# B&R Automation Studio project AP124
Automation Studio 4.2.8.54 SP; technology packages: mapp 1.40.0, TextSystem 

## Configuration CP1583

CPU X20CP1583, AutomationRuntime A4.26, Build 4.1.2, Vc V4.26.1, Safety 1.9

### Task classes (Cpu.sw)
```
Cyclic#3 (cycle 50000 us, tolerance 50000 us):
  pallet_mag <- plc.pallet_magazine.pallet_magazine.prg
  pallet_con <- plc.palletization.pallet_conveyors.pallet_conveyors.prg
  product_in <- plc.palletization.product_infeed.product_infeed.prg
  robot_head <- plc.palletization.robot_head.robot_head.prg
  robot_cont <- plc.palletization.robot_control.robot_control.prg
  wrapper <- plc.pallet_outfeed.wrapper.wrapper.prg
  pallet_out <- plc.pallet_outfeed.pallet_outfeed.pallet_outfeed.prg
  alarm_mana <- plc.alarm_management.alarm_management.prg
  safety <- safety.safety.prg
Cyclic#4 (cycle 100000 us, tolerance 100000 us):
  visu_manag <- visualization.visu_manager.prg
  visu_roman <- visualization.visu_roman.prg
DataObjects: assl1
VcDataObjects: Visu <- visualization.Visu.dob
Binaries: TCData, vcctext, arialbd, vcmgr, vccshape, vcnet, Visu02, vcbclass, vcfntttf, vctcal, Visu03, vcshared, vcrt, vcpkat, Visu01, vccbmp, vcfile, vccbtn, vccdt, vcalarm, vccnum, vcchspot, vcpdsw, vcdsint, arial, vccovl, udbdef, vccline, vcpdvnc, vccalarm, vccstr, vcchtml, vcxml, vcgclass, vccurl, vcdsloc, vcpfx20, sysconf, ashwd, asfw, iomap, Role, User, arconfig, TC, vcclbox, vcpfar00, vccscale, vccslider, arsvcreg
Libraries: AsSafety, FileIO, AsXml, standard, runtime, astime, asieccon, asstring, ashw, dataobj, vcresman, MTBasics, brsystem, MTTypes, sys_lib, AsBrStr, AcpInoSdc, AsIOAcc, AsBrMath, AsEPL, visapi
```

### Hardware
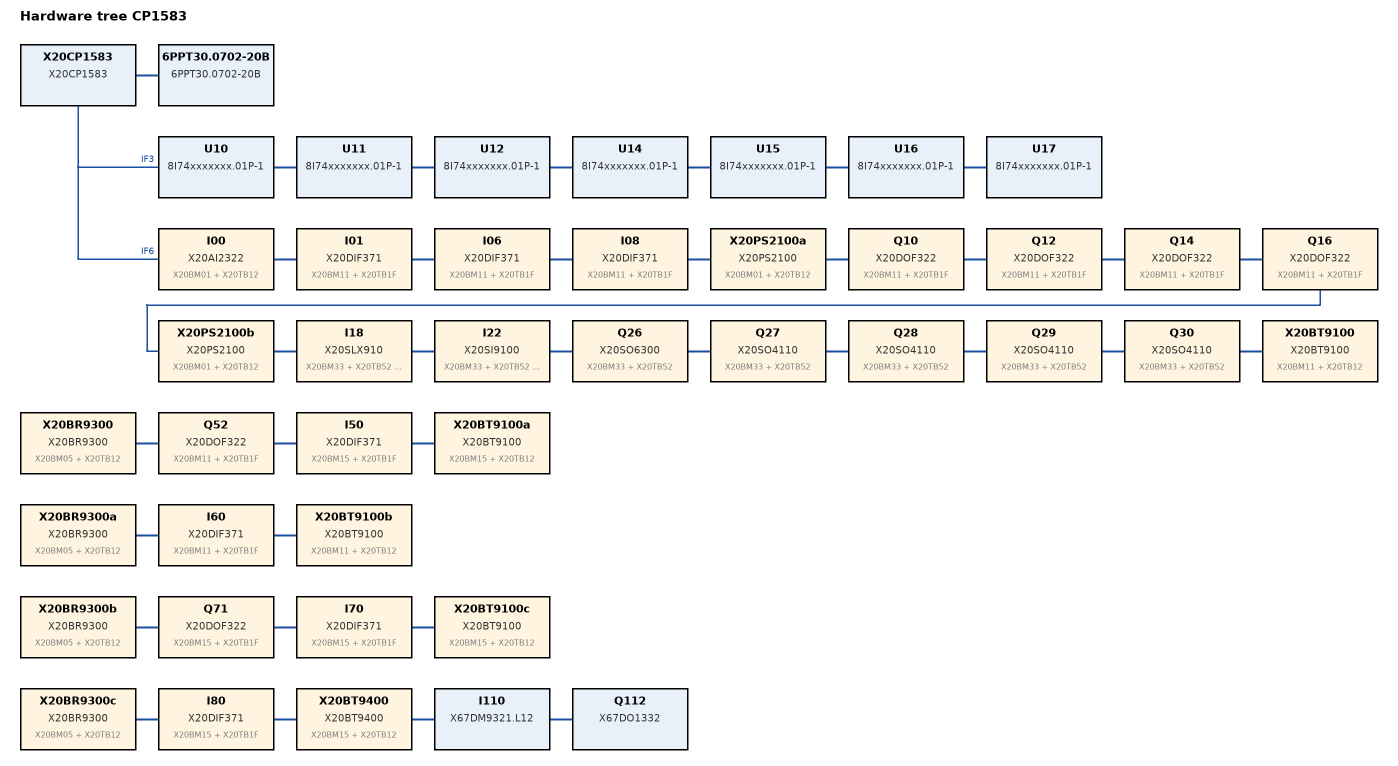
```
6PPT30.0702-20B : 6PPT30.0702-20B v1.1.0.0  [ETH1 -> X20CP1583.IF2 (NodeNumber=1)]
  Terminal = true
  Startmode = 1
  Mode = Manual
  InternetAddress = 192.168.88.11
  DefaultGateway = 192.168.88.1
  Subnetmask = 255.255.255.0
  ActivateOpenService = 0
  SelectedFavoriteVNC = 192.168.88.10
  PasswordVNC = 
  PasswordCIFS = 
  PasswordService = 
I00 : X20AI2322 v1.0.0.2  [SS1 -> X20TB12.SS; SL -> X20BM01.SL1]
  ChannelType01 = 4 to 20mA
I01 : X20DIF371 v1.0.1.0  [SS1 -> X20TB1F12.SS; SL -> X20BM11q.SL1]
I06 : X20DIF371 v1.0.1.0  [SS1 -> X20TB1F.SS; SL -> X20BM11.SL1]
I08 : X20DIF371 v1.0.1.0  [SS1 -> X20TB1F1.SS; SL -> X20BM11a.SL1]
I110 : X67DM9321.L12 v1.1.1.1 (Disabled=true)  [X2X1 -> X20BT9400.X2X1 (NodeNumber=33)]
I18 : X20SLX910 v1.10.0.0  [SS1 -> X20TB52.SS; SS2 -> X20TB52a.SS; SL -> X20BM33.SL1]
  SafeProject = SafeLOGIC-1
  SafeDesigner = 4.2.0.17
  UnsafeOutputBOOLs = 24
  UnsafeInputBOOLs = 24
I22 : X20SI9100 v1.10.0.1  [SS1 -> X20TB52b.SS; SS2 -> X20TB52c.SS; SL -> X20BM33a.SL1]
I50 : X20DIF371 v1.0.1.0  [SS1 -> X20TB1F6.SS; SL -> X20BM15f.SL1]
I60 : X20DIF371 v1.0.1.0  [SS1 -> X20TB1F8.SS; SL -> X20BM11j.SL1]
I70 : X20DIF371 v1.0.1.0  [SS1 -> X20TB1F9.SS; SL -> X20BM15c.SL1]
I80 : X20DIF371 v1.0.1.0  [SS1 -> X20TB1F11.SS; SL -> X20BM15a.SL1]
Q10 : X20DOF322 v1.1.0.2  [SS1 -> X20TB1F2.SS; SL -> X20BM11b.SL1]
Q112 : X67DO1332 v1.0.0.2 (Disabled=true)  [X2X1 -> I110.X2X2]
Q12 : X20DOF322 v1.1.0.2  [SS1 -> X20TB1F3.SS; SL -> X20BM11c.SL1]
Q14 : X20DOF322 v1.1.0.2  [SS1 -> X20TB1F4.SS; SL -> X20BM11d.SL1]
Q16 : X20DOF322 v1.1.0.2  [SS1 -> X20TB1F5.SS; SL -> X20BM11e.SL1]
Q26 : X20SO6300 v1.10.0.1  [SS1 -> X20TB52d.SS; SL -> X20BM33b.SL1]
  SafeModuleID = 3
  DigitalOutput01 = viaSafeLOGIC
  DigitalOutput02 = viaSafeLOGIC
  DigitalOutput03 = viaSafeLOGIC
  DigitalOutput04 = viaSafeLOGIC
  DigitalOutput05 = viaSafeLOGIC
  DigitalOutput06 = viaSafeLOGIC
Q27 : X20SO4110 v1.10.0.1  [SS1 -> X20TB52e.SS; SL -> X20BM33c.SL1]
  SafeModuleID = 4
Q28 : X20SO4110 v1.10.0.1  [SS1 -> X20TB52f.SS; SL -> X20BM33d.SL1]
  SafeModuleID = 5
Q29 : X20SO4110 v1.10.0.1  [SS1 -> X20TB52g.SS; SL -> X20BM33e.SL1]
  SafeModuleID = 6
  DigitalOutput01 = viaSafeLOGIC
  DigitalOutput02 = viaSafeLOGIC
  DigitalOutput03 = viaSafeLOGIC
  DigitalOutput04 = viaSafeLOGIC
Q30 : X20SO4110 v1.10.0.1  [SS1 -> X20TB52h.SS; SL -> X20BM33f.SL1]
  SafeModuleID = 7
  DigitalOutput01 = viaSafeLOGIC
  DigitalOutput02 = viaSafeLOGIC
  DigitalOutput03 = viaSafeLOGIC
  DigitalOutput04 = viaSafeLOGIC
Q52 : X20DOF322 v1.1.0.2  [SS1 -> X20TB1F7.SS; SL -> X20BM11h.SL1]
Q71 : X20DOF322 v1.1.0.2  [SS1 -> X20TB1F10.SS; SL -> X20BM15d.SL1]
U10 : 8I74xxxxxxx.01P-1 v1.3.0.0  [PLK1 -> X20CP1583.IF3 (NodeNumber=10); PLK2 -> U11.PLK1 (NodeNumber=10)]
  Supervision = off
  packedETAD = packed
  packedETI = packed
  packedCMDD = packed
  packedCMI = packed
  ACC = 5
  DEC = 3
  HSP = 600
  NPR = 55
  COS = 72
  UNS = 400
  NCR = 16
  NSP = 1360
  BLC = 2
  BST = 0
U11 : 8I74xxxxxxx.01P-1 v1.3.0.0  [PLK1 -> U10.PLK2 (NodeNumber=11); PLK2 -> U12.PLK1 (NodeNumber=11)]
  Supervision = off
  packedETAD = packed
  packedETI = packed
  packedCMDD = packed
  packedCMI = packed
  ACC = 5
  DEC = 5
  HSP = 600
  NPR = 55
  COS = 72
  UNS = 400
  NCR = 16
  NSP = 1360
  BLC = 2
  BST = 0
U12 : 8I74xxxxxxx.01P-1 v1.3.0.0  [PLK1 -> U11.PLK2 (NodeNumber=12); PLK2 -> U14.PLK1 (NodeNumber=12)]
  Supervision = off
  packedETAD = packed
  packedETI = packed
  packedCMDD = packed
  packedCMI = packed
  ACC = 0
  DEC = 0
  FLU = 0
  NPR = 110
  COS = 73
  UNS = 400
  NCR = 26
  NSP = 1455
  RSA = 4824
  LFA = 4327
  IDA = 19
  TRA = 153
  ADC = 0
U14 : 8I74xxxxxxx.01P-1 v1.3.0.0  [PLK1 -> U12.PLK2 (NodeNumber=14); PLK2 -> U15.PLK1 (NodeNumber=14)]
  Supervision = off
  packedETAD = packed
  packedETI = packed
  packedCMDD = packed
  packedCMI = packed
  LFRD_LFR_Filter = LFR_RFR
  ACC = 5
  DEC = 5
  HSP = 600
  NPR = 55
  COS = 72
  UNS = 400
  NCR = 16
  NSP = 1360
  BLC = 2
  BST = 0
U15 : 8I74xxxxxxx.01P-1 v1.3.0.0  [PLK1 -> U14.PLK2 (NodeNumber=15); PLK2 -> U16.PLK1 (NodeNumber=15)]
  Supervision = off
  packedETAD = packed
  packedETI = packed
  packedCMDD = packed
  packedCMI = packed
  LFRD_LFR_Filter = LFR_RFR
  ACC = 5
  DEC = 5
  HSP = 600
  NPR = 55
  COS = 72
  UNS = 400
  NCR = 16
  NSP = 1360
U16 : 8I74xxxxxxx.01P-1 v1.3.0.0  [PLK1 -> U15.PLK2 (NodeNumber=16); PLK2 -> U17.PLK1 (NodeNumber=16)]
  Supervision = off
  packedETAD = packed
  packedETI = packed
  packedCMDD = packed
  packedCMI = packed
  LFRD_LFR_Filter = LFR_RFR
  ACC = 5
  DEC = 5
  HSP = 600
  NPR = 55
  COS = 72
  UNS = 400
  NCR = 16
  NSP = 1360
U17 : 8I74xxxxxxx.01P-1 v1.3.0.0  [PLK1 -> U16.PLK2 (NodeNumber=17)]
  Supervision = off
  packedETAD = packed
  packedETI = packed
  packedCMDD = packed
  packedCMI = packed
  LFRD_LFR_Filter = LFR_RFR
  ACC = 5
  DEC = 5
  HSP = 600
  NPR = 55
  COS = 72
  UNS = 400
  NCR = 16
  NSP = 1360
X20BM01 : X20BM01 v1.0.1.1  [X2X1 -> X20CP1583.IF6]
X20BM01a : X20BM01 v1.0.1.1  [X2X1 -> X20BM11a.X2X2]
X20BM01b : X20BM01 v1.0.1.1  [X2X1 -> X20BM11e.X2X2]
X20BM05 : X20BM05 v1.0.0.3
X20BM05a : X20BM05 v1.0.0.3
X20BM05b : X20BM05 v1.0.0.3
X20BM05c : X20BM05 v1.0.0.3
X20BM11 : X20BM11 v1.0.0.1  [X2X1 -> X20BM11q.X2X2]
X20BM11a : X20BM11 v1.0.0.1  [X2X1 -> X20BM11.X2X2]
X20BM11b : X20BM11 v1.0.0.1  [X2X1 -> X20BM01a.X2X2]
X20BM11c : X20BM11 v1.0.0.1  [X2X1 -> X20BM11b.X2X2]
X20BM11d : X20BM11 v1.0.0.1  [X2X1 -> X20BM11c.X2X2]
X20BM11e : X20BM11 v1.0.0.1  [X2X1 -> X20BM11d.X2X2]
X20BM11f : X20BM11 v1.0.0.1  [X2X1 -> X20BM33f.X2X2]
X20BM11h : X20BM11 v1.0.0.1  [X2X1 -> X20BM05.X2X2]
X20BM11j : X20BM11 v1.0.0.1  [X2X1 -> X20BM05a.X2X2]
X20BM11k : X20BM11 v1.0.0.1  [X2X1 -> X20BM11j.X2X2]
X20BM11q : X20BM11 v1.0.0.1  [X2X1 -> X20BM01.X2X2]
X20BM15 : X20BM15 v1.0.1.0  [X2X1 -> X20BM15a.X2X2 (NodeNumber=32)]
X20BM15a : X20BM15 v1.0.1.0  [X2X1 -> X20BM05c.X2X2 (NodeNumber=31)]
X20BM15b : X20BM15 v1.0.1.0  [X2X1 -> X20BM15c.X2X2 (NodeNumber=29)]
X20BM15c : X20BM15 v1.0.1.0  [X2X1 -> X20BM15d.X2X2 (NodeNumber=28)]
X20BM15d : X20BM15 v1.0.1.0  [X2X1 -> X20BM05b.X2X2 (NodeNumber=27)]
X20BM15e : X20BM15 v1.0.1.0  [X2X1 -> X20BM15f.X2X2 (NodeNumber=22)]
X20BM15f : X20BM15 v1.0.1.0  [X2X1 -> X20BM11h.X2X2 (NodeNumber=21)]
X20BM33 : X20BM33 v1.0.0.4  [X2X1 -> X20BM01b.X2X2]
X20BM33a : X20BM33 v1.0.0.4  [X2X1 -> X20BM33.X2X2]
X20BM33b : X20BM33 v1.0.0.4  [X2X1 -> X20BM33a.X2X2]
X20BM33c : X20BM33 v1.0.0.4  [X2X1 -> X20BM33b.X2X2]
X20BM33d : X20BM33 v1.0.0.4  [X2X1 -> X20BM33c.X2X2]
X20BM33e : X20BM33 v1.0.0.4  [X2X1 -> X20BM33d.X2X2]
X20BM33f : X20BM33 v1.0.0.4  [X2X1 -> X20BM33e.X2X2]
X20BR9300 : X20BR9300 v1.0.3.0  [SS1 -> X20TB12d.SS; SL -> X20BM05.SL1; X2X1 -> X20BT9100.X2X1 (NodeNumber=19)]
X20BR9300a : X20BR9300 v1.0.3.0  [SS1 -> X20TB12g.SS; SL -> X20BM05a.SL1; X2X1 -> X20BT9100a.X2X1 (NodeNumber=23)]
X20BR9300b : X20BR9300 v1.0.3.0  [SS1 -> X20TB12i.SS; SL -> X20BM05b.SL1; X2X1 -> X20BT9100b.X2X1 (NodeNumber=26)]
X20BR9300c : X20BR9300 v1.0.3.0  [SS1 -> X20TB12l.SS; SL -> X20BM05c.SL1; X2X1 -> X20BT9100c.X2X1 (NodeNumber=30)]
X20BT9100 : X20BT9100 v1.0.2.4  [SS1 -> X20TB12c.SS; SL -> X20BM11f.SL1]
X20BT9100a : X20BT9100 v1.0.2.4  [SS1 -> X20TB12f.SS; SL -> X20BM15e.SL1]
X20BT9100b : X20BT9100 v1.0.2.4  [SS1 -> X20TB12h.SS; SL -> X20BM11k.SL1]
X20BT9100c : X20BT9100 v1.0.2.4  [SS1 -> X20TB12k.SS; SL -> X20BM15b.SL1]
X20BT9400 : X20BT9400 v1.0.1.4  [SS1 -> X20TB12m.SS; SL -> X20BM15.SL1]
X20CP1583 : X20CP1583 v1.3.0.0
  Connector IF2:
    ActivateDevice = 1
    EthInterfaceRedundant = 0
    Mode = Manual
    InternetAddress = 192.168.88.10
    SubnetMask = 255.255.255.0
    Vnc1
    VncVcObjectName1 = Visu
    VncKeyMappingFile1 = VC\PS2-Keyboard1.dis
    VncMaxConnections1 = 2
    VncRefreshRate1 = 100
  Connector IF3:
    EplInterfaceRedundant = 0
    EplEthInterfaceRedundant = 0
  ConfigurationID = AP124_CP1583
  UserPartitionSize = 200
  Simulation = 1
  VolatileGlobalPvSize = 262144
  TimerDeviceType = EPLX2X
  TimerDevice = X20CP1583.IF3
  TaskClassIdleTime = 2000
  Cyclic1Duration = 10000
  Cyclic1Tolerance = 10000
  Cyclic1Output = 1
  Cyclic2Duration = 20000
  Cyclic2Tolerance = 20000
  Cyclic3Duration = 50000
  Cyclic3Tolerance = 50000
  Cyclic4Duration = 100000
  Cyclic4Tolerance = 100000
  Cyclic5Duration = 200000
  Cyclic5Tolerance = 200000
  Cyclic6Duration = 500000
  Cyclic6Tolerance = 500000
  Cyclic7Duration = 1000000
  Cyclic7Tolerance = 1000000
  Cyclic8Duration = 10000
  Cyclic8Tolerance = 30000000
  FileDevice1
  FileDeviceName1 = USER
  FileDevicePath1 = F:\
  FtpUser1
  FtpUsername1 = atrima
  FtpUserPassword1 = WTu4FPCiIceACZRqUEgJEtXb7Eb63HUzCfqgyyypU7s=
  FtpUserSalt1 = 2eJIzixw
  FTPAccessRight1 = 0
X20PS2100a : X20PS2100 v1.1.0.0  [SS1 -> X20TB12a.SS; SL -> X20BM01a.SL1]
X20PS2100b : X20PS2100 v1.1.0.0  [SS1 -> X20TB12b.SS; SL -> X20BM01b.SL1]
X20TB12 : X20TB12 v1.0.0.0
X20TB12a : X20TB12 v1.0.0.0
X20TB12b : X20TB12 v1.0.0.0
X20TB12c : X20TB12 v1.0.0.0
X20TB12d : X20TB12 v1.0.0.0
X20TB12f : X20TB12 v1.0.0.0
X20TB12g : X20TB12 v1.0.0.0
X20TB12h : X20TB12 v1.0.0.0
X20TB12i : X20TB12 v1.0.0.0
X20TB12k : X20TB12 v1.0.0.0
X20TB12l : X20TB12 v1.0.0.0
X20TB12m : X20TB12 v1.0.0.0
X20TB1F : X20TB1F v1.0.0.0
X20TB1F1 : X20TB1F v1.0.0.0
X20TB1F10 : X20TB1F v1.0.0.0
X20TB1F11 : X20TB1F v1.0.0.0
X20TB1F12 : X20TB1F v1.0.0.0
X20TB1F2 : X20TB1F v1.0.0.0
X20TB1F3 : X20TB1F v1.0.0.0
X20TB1F4 : X20TB1F v1.0.0.0
X20TB1F5 : X20TB1F v1.0.0.0
X20TB1F6 : X20TB1F v1.0.0.0
X20TB1F7 : X20TB1F v1.0.0.0
X20TB1F8 : X20TB1F v1.0.0.0
X20TB1F9 : X20TB1F v1.0.0.0
X20TB52 : X20TB52 v1.0.0.1
X20TB52a : X20TB52 v1.0.0.1
X20TB52b : X20TB52 v1.0.0.1
X20TB52c : X20TB52 v1.0.0.1
X20TB52d : X20TB52 v1.0.0.1
X20TB52e : X20TB52 v1.0.0.1
X20TB52f : X20TB52 v1.0.0.1
X20TB52g : X20TB52 v1.0.0.1
X20TB52h : X20TB52 v1.0.0.1
```

### IoMap.iom - X20CP1583/IoMap.iom
(iom body not rendered)

### Acp10cfg.ncc - X20CP1583/Motion/Acp10cfg.ncc
```
NcConfiguration (Version=3.13.0, NcSwId=Acp10)
  ACP10CF1_typ:
    cnt_nettrc_rec_drive = 1500
    bufsize_trace_upload = 1200
    tc_nc_man_task = Cyclic #1
    glob_pv_as_ncobject = Yes
    ncsys_dl_broadcast = Yes
    ncsys_dl_acp_reset = Yes
    safemc_log_err_to_ax = Yes
    network_init:
      ncsw_init_execute = Yes
      automatic_execute = No
      node_nr_warning = Yes
      net_err_before_ncact = Yes
    nettrc:
      enter_parsecrec = Yes
      enter_ncaction = Yes
      save_ring_startidx = Yes
    cam_prof_download:
      cam_dat_dl_parallel = No
      tc_cam_dl_parallel = Task class for NC Manager task
    sdc_if[0]:
      if_name = SDC_IF1
      mc_broadcast_size = 800
      mc_broadcast_extdat = No
```

### Acp10map.ncm - X20CP1583/Motion/Acp10map.ncm
```
NcMapping (NcSwId=Acp10)
  NcObject U15a_ncAXIS1 (ModuleId=U16, ModuleAddress=SDC_IF1.ST1, Type=ncAXIS, Channel=1, AcoposSimulation=Off, Disabled=TRUE, ModuleDisabled=FALSE)
  NcObject U15b_ncAXIS1 (ModuleId=U17, ModuleAddress=SDC_IF1.ST2, Type=ncAXIS, Channel=1, AcoposSimulation=Off, Disabled=TRUE, ModuleDisabled=FALSE)
```

- Safety project (password-protected, skipped)

### Config.mprecipecsv - X20CP1583/mapp/Config.mprecipecsv
```
Element gRecipeCsv (Type=mprecipecsv)
```

### Config_1.mpalarmxcore - X20CP1583/mapp/Config_1.mpalarmxcore
```
Element gAlarmXCore (Type=mpalarmxcore)
  mapp.AlarmX.Core.Configuration:
    [0]:
      Name = AirPressureNotOK
      Message = Air pressure not OK
      Behavior = PersistentAlarm
    [1]:
      Name = MagazineUpperHwEndReached
      Message = Magazine upper HW end reached
      Behavior:
        MultipleInstances = FALSE
    [2]:
      Name = MagazineLooseChain
      Message = Magazine loose chain
      Behavior:
        MultipleInstances = FALSE
    [3]:
      Name = MotorProtectionP11
      Message = Motor protection P11 failure
      Behavior = PersistentAlarm
    [4]:
      Name = EStop1
      Message = E-Stop 1
    [5]:
      Name = EStop1
      Message = E-Stop 1
    [6]:
      Name = EStop3
      Message = E-Stop 3
      Behavior = PersistentAlarm
    [7]:
      Name = EStop4
      Message = E-Stop 4
      Behavior = PersistentAlarm
    [8]:
      Name = EStop5
      Message = E-Stop 5
      Behavior = PersistentAlarm
    [9]:
      Name = EStopRobot
      Message = E-Stop Robot
      Behavior = PersistentAlarm
    [10]:
      Name = EStopWrapper
      Message = E-Stop Wrapper
      Behavior = PersistentAlarm
```

## Logical view

Binary libraries used (declarations not repeated): operator, runtime, astime, AsIecCon, AsSafety, FileIO, AsXml, standard, asstring, MTBasics 2.20.0, brsystem, MTTypes 1.03.0, sys_lib, AsBrStr, AsIOAcc, AsBrMath, AsEPL, visapi, MpCom 1.40.0, MpRecipe 1.40.0, AsIODiag, MpAlarmX 1.30.0

- VST_VYST_PROG.xlsx - přiřazení vstupů a výstupů (binary file, 31416 bytes)
- AP124 documentation.odt (binary file, 12845 bytes)
### Global.var - Global variables
```iecst
VAR
	RecipeChanged : BOOL;
END_VAR
```

### Package Logical/Libraries - Global libraries

### Library Logical/Libraries/AcpInoSdc (IEC)

#### AcpInoSdc.fun - Exported functions and function blocks
```iecst
FUNCTION_BLOCK AcpInoSdc (*control of ACOPOSinverter without SDC*) (*$GROUP=User,$CAT=User,$GROUPICON=User.png,$CATICON=User.png*)
	VAR_INPUT
		switchOn : BOOL;
		quickStop : BOOL;
		reset : BOOL := TRUE;
		speed : INT;
		ETAD_Input : UINT;
		run : BOOL := TRUE;
	END_VAR
	VAR_OUTPUT
		CMDD_Output : UINT;
		LFRD_Output : INT;
		switchedOn : BOOL;
		error : BOOL;
	END_VAR
END_FUNCTION_BLOCK
```

#### AcpInoSdc.st
```iecst
(* control of ACOPOSinverter without SDC *)
FUNCTION_BLOCK AcpInoSdc

	LFRD_Output := speed;

	CASE ETAD_Input AND 16#FF  OF
		16#40, 16#50: (* Switch on disabled *)
		CMDD_Output := 16#0006;

		16#21, 16#31: (*Ready to switch on *)
		IF switchOn THEN
			CMDD_Output := 16#0007;
		END_IF

		16#33, 16#23: (*Switched on *)
		CMDD_Output := 16#000F;

		16#37, 16#27: (*Operation enabled *)
		IF stop THEN
//			LFRD_Output := 0;
			CMDD_Output := 16#010F;
		ELSE
			CMDD_Output := 16#000F;
		END_IF

		IF NOT switchOn THEN
			CMDD_Output := 16#0006;
		END_IF

		IF quickStop THEN
			CMDD_Output := 16#0002;
		END_IF

		16#17, 16#07: (*Quick stop active *)
		quickStop := FALSE;
		switchOn := FALSE;
		CMDD_Output := 16#0000;
	END_CASE;

	(* Fault *)
	error := ETAD_Input.3 OR ETAD_Input = 0;
//
//	IF 	DiagCpuIsSimulated() THEN
//		error := FALSE;
//	END_IF

	IF reset AND ETAD_Input.3 THEN
		CMDD_Output := 16#0080;
	END_IF
	reset := FALSE;

	switchedOn := ETAD_Input.1;
END_FUNCTION_BLOCK
```

### Library Logical/Libraries/Motorky (ANSIC, version 2.20.0)

#### Motorky.typ
```iecst
TYPE
	Motorky_ActualSpeed : 	STRUCT
		actPosition : DINT;
		actSpeed : DINT;
		taskTime : DINT;
		filterTime : DINT;
		positionDifference : DINT;
		FIFOsize : DINT;
		FIFOindex : DINT;
		positionFIFO : ARRAY[0..SPEED_FIFO_UBOUND]OF DINT;
	END_STRUCT;
	Motorky_Cmd_typ : 	STRUCT
		power : BOOL;
		homing : BOOL;
		absolute : BOOL;
		additive : BOOL;
		cyclicPosition : BOOL;
		velocity : BOOL;
		acknowledge : BOOL;
		stop : BOOL;
	END_STRUCT;
	Motorky_ConvertAcceleration : 	STRUCT
		inputScale : DINT;
		outputScale : DINT;
		maxAcceleration : DINT;
		status : UINT;
	END_STRUCT;
	Motorky_ConvertPosition : 	STRUCT
		inputScale : DINT;
		outputScale : DINT;
		reverseDirection : BOOL;
		input : INT;
		output : DINT;
		dInput : INT;
		integral : DINT;
	END_STRUCT;
	Motorky_ConvertSpeed : 	STRUCT
		inputScale : DINT;
		outputScale : DINT;
		maxSpeed : DINT;
		status : UINT;
	END_STRUCT;
	Motorky_DS_Intern_typ : 	STRUCT
		step : UINT;
		oldStep : UINT;
		oldPosition : DINT;
		oldReferenceSwitch : BOOL;
		movTargetTimeOffset : DINT;
		pathGenerator : Motorky_PathGenerator;
		convertPosition : Motorky_ConvertPosition;
		actualSpeed : Motorky_ActualSpeed;
	END_STRUCT;
	Motorky_DS_IOMapping : 	STRUCT
		DriveReady : BOOL;
		SystemTime : DINT;
		DriveEnable : BOOL;
		MovTargetTime : DINT;
		MovTargetPosition : DINT;
		positiveLimitSwitch : BOOL;
		negativeLimitSwitch : BOOL;
		referenceSwitch : BOOL;
	END_STRUCT;
	Motorky_FI_IOMapping : 	STRUCT
		DriveReady : BOOL;
		Encoder : INT;
		DriveEnable : BOOL;
		AnalogOutput : INT;
		positiveLimitSwitch : BOOL;
		negativeLimitSwitch : BOOL;
		referenceSwitch : BOOL;
	END_STRUCT;
	Motorky_Info_typ : 	STRUCT
		initialized : BOOL;
		powerOn : BOOL;
		homingOk : BOOL;
		position : DINT;
		speed : DINT;
		moveActive : BOOL;
		lagError : DINT;
		status : UINT;
		errorText : STRING[100];
	END_STRUCT;
	Motorky_Init_MM_typ : 	STRUCT
		taskTime : REAL;
		units : DINT;
		encoderIncrements : DINT;
		reverseDirection : BOOL;
		maxLagError : DINT;
		Kp : REAL;
		Tn : REAL;
		speedKp : REAL;
		speedTn : REAL;
		speedFilter : REAL;
		settleTime : REAL;
		positiveSwLimit : DINT;
		negativeSwLimit : DINT;
	END_STRUCT;
	Motorky_Init_Enc_typ : 	STRUCT
		taskTime : REAL;
		units : DINT;
		encoderIncrements : DINT;
		reverseDirection : BOOL;
		maxLagError : DINT;
		Kp : REAL;
		Tn : REAL;
		speedFilter : REAL;
		settleTime : REAL;
		positiveSwLimit : DINT;
		negativeSwLimit : DINT;
	END_STRUCT;
	Motorky_Init_SM_typ : 	STRUCT
		taskTime : REAL;
		units : DINT;
		microsteps : DINT;
		reverseDirection : BOOL;
		settleTime : REAL;
		positiveSwLimit : DINT;
		negativeSwLimit : DINT;
		outputFilter : REAL;
	END_STRUCT;
	Motorky_Init_NoEnc_typ : 	STRUCT
		taskTime : REAL;
		units : DINT;
		microsteps : DINT;
		reverseDirection : BOOL;
		settleTime : REAL;
		positiveSwLimit : DINT;
		negativeSwLimit : DINT;
	END_STRUCT;
	Motorky_Intern_typ : 	STRUCT
		step : UINT;
		oldStep : UINT;
		oldPosition : DINT;
		oldReferenceSwitch : BOOL;
		pathGenerator : Motorky_PathGenerator;
		moveActive : Motorky_MoveActive;
	END_STRUCT;
	Motorky_InternFI_typ : 	STRUCT
		encoder2units : Motorky_ConvertPosition;
		pid : Motorky_PID;
		actualSpeed : Motorky_ActualSpeed;
	END_STRUCT;
	Motorky_InternMM_typ : 	STRUCT
		encoder2units : Motorky_ConvertPosition;
		pid : Motorky_PID;
		actualSpeed : Motorky_ActualSpeed;
		speedPID : Motorky_PID;
	END_STRUCT;
	Motorky_MM_Intern_typ : 	STRUCT
		step : UINT;
		oldStep : UINT;
		encoderPosition : INT;
		oldPosition : DINT;
		oldReferenceSwitch : BOOL;
		pathGenerator : Motorky_PathGenerator;
		convertPosition : Motorky_ConvertPosition;
		actualSpeed : Motorky_ActualSpeed;
		moveActive : Motorky_MoveActive;
		pid : Motorky_PID;
	END_STRUCT;
	Motorky_MM_IOMapping : 	STRUCT
		DriveReady : BOOL;
		DriveEnable : BOOL;
		PeriodDuration : UINT;
		PulseWidth : INT;
		ClearError : BOOL;
		Counter : INT;
		UnderVoltageError : BOOL;
		OverVoltageError : BOOL;
		OvertemperatureError : BOOL;
		OvercurrentError : BOOL;
		positiveLimitSwitch : BOOL;
		negativeLimitSwitch : BOOL;
		referenceSwitch : BOOL;
	END_STRUCT;
	Motorky_MoveActive : 	STRUCT
		motionState : UINT;
		taskTime : DINT;
		settleTime : DINT;
		settleTimer : DINT;
		moveActive : BOOL;
	END_STRUCT;
	Motorky_OutputGenerator : 	STRUCT
		enable : BOOL;
		encoderUsed : BOOL;
		reverseDirection : BOOL;
		setPosition : DINT;
		actPosition : DINT;
		setSpeed : DINT;
		motionState : UINT;
		settleTime : DINT;
		Y : DINT;
		moveActive : BOOL;
		settleTimer : DINT;
		taskTime : DINT;
		e : DINT;
		Kp : DINT;
		Ki : DINT;
		Yp : DINT;
		Yi : DINT;
		Yiintegral : DINT;
	END_STRUCT;
	Motorky_Param_Homing : 	STRUCT
		mode : USINT;
		startDirection : BOOL;
		edgeSwitch : BOOL;
		triggerDirection : BOOL;
		speed2 : DINT;
	END_STRUCT;
	Motorky_Param_typ : 	STRUCT
		position : DINT;
		speed : DINT;
		acceleration : DINT;
		deceleration : DINT;
		homing : Motorky_Param_Homing;
	END_STRUCT;
	Motorky_PathGenerator : 	STRUCT
		moveCommand : USINT;
		setPosition : DINT;
		setSpeed : DINT;
		acceleration : DINT;
		deceleration : DINT;
		positiveSwLimit : DINT;
		negativeSwLimit : DINT;
		outputPosition : DINT;
		outputSpeed : DINT;
		motionState : UINT;
		status : UINT;
		step : UINT;
		speedRamping : Motorky_SpeedRamping;
	END_STRUCT;
	Motorky_PID : 	STRUCT
		enable : BOOL;
		W : DINT;
		X : DINT;
		Y : DINT;
		Kp : DINT;
		Y_max : DINT;
		Y_min : DINT;
		e : DINT;
		Yp : DINT;
		Yi : DINT;
		Yi_sum : DINT;
		Ki : DINT;
		Ytotal : DINT;
		Ylim : DINT;
		Ywindup : DINT;
	END_STRUCT;
	Motorky_SM_Intern_typ : 	STRUCT
		step : UINT;
		oldStep : UINT;
		setPosition : DINT;
		oldPosition : DINT;
		dPosition : DINT;
		oldReferenceSwitch : BOOL;
		pathGenerator : Motorky_PathGenerator;
		outputConversion : Motorky_ConvertPosition;
		actualSpeed : Motorky_ActualSpeed;
		tofBoostCurrent : Motorky_TOF;
		moveActive : Motorky_MoveActive;
	END_STRUCT;
	Motorky_SM_IOMapping : 	STRUCT
		DriveReady : BOOL;
		MotorStep0 : INT;
		DriveEnable : BOOL;
		BoostCurrent : BOOL;
		StandstillCurrent : BOOL;
		StallError : BOOL;
		OvertemperatureError : BOOL;
		OvercurrentError : BOOL;
		ModulePowerSupplyError : BOOL;
		ClearError : BOOL;
		UZKStatus : BOOL;
		positiveLimitSwitch : BOOL;
		negativeLimitSwitch : BOOL;
		referenceSwitch : BOOL;
	END_STRUCT;
	Motorky_SpeedRamping : 	STRUCT
		setSpeed : DINT;
		acceleration : DINT;
		deceleration : DINT;
		actualPosition : DINT;
		actualSpeed : DINT;
		motionState : UINT;
		divisor : DINT;
		sIntegral : DINT;
		vIntegral : DINT;
	END_STRUCT;
	Motorky_TOF : 	STRUCT
		IN : BOOL;
		PT : DINT;
		Q : BOOL;
		ET : DINT;
	END_STRUCT;
END_TYPE
```

#### Motorky.var
```iecst
VAR CONSTANT
	MOVE_COMMAND_STOP : USINT := 0;
	HOMING_DIRECT : USINT := 0;
	MOTION_STATE_STANDSTILL : UINT := 0;
	DIRECTION_POSITIVE : UINT := 0;
	MOTION_STATE_ACCELERATING : UINT := 1;
	HOMING_END_SWITCH : USINT := 1;
	MOVE_COMMAND_ABSOLUTE : USINT := 1;
	DIRECTION_NEGATIVE : UINT := 1;
	MOVE_COMMAND_VELOCITY : USINT := 2;
	MOTION_STATE_CONSTANT_SPEED : UINT := 2;
	HOMING_REF_SWITCH : USINT := 2;
	MOTION_STATE_DECELERATING : UINT := 3;
	ERR_CONTROLLER_OFF : UINT := 40001;
	ERR_WRONG_UNITS : UINT := 40002;
	ERR_NEGATIVE_LIMIT_SWITCH_CLOSED : UINT := 40003;
	ERR_NEGATIVE_SW_LIMIT_REACHED : UINT := 40004;
	ERR_OVER_CURRENT : UINT := 40006;
	ERR_OVER_TEMPERATURE : UINT := 40007;
	ERR_POSITIVE_LIMIT_SWITCH_CLOSED : UINT := 40008;
	ERR_POSITIVE_SW_LIMIT_REACHED : UINT := 40009;
	ERR_STALL : UINT := 40011;
	ERR_DRIVE_NOT_READY : UINT := 40012;
	ERR_POWER_SUPPLY_ERROR : UINT := 40013;
	ERR_UNDER_VOLTAGE : UINT := 40014;
	ERR_OVER_VOLTAGE : UINT := 40015;
	ERR_LAG_ERROR : UINT := 40016;
	ERR_ENCODER_SUPPLY : UINT := 40017;
	ERR_WRONG_TASK_TIME : UINT := 40018;
	ERR_LOW_DC_BUS_VOLTAGE : UINT := 40019;
	ERR_WRONG_ENCODER_INCREMENTS : UINT := 40020;
	ERR_DRV_NOT_OK : UINT := 40021;
	SPEED_FIFO_UBOUND : INT := 19;
END_VAR
```

#### Motorky.fun
```iecst
FUNCTION_BLOCK FI
	VAR_INPUT
		init : Motorky_Init_Enc_typ;
		cmd : Motorky_Cmd_typ;
		param : Motorky_Param_typ;
	END_VAR
	VAR_OUTPUT
		info : Motorky_Info_typ;
		IOMapping : Motorky_FI_IOMapping;
	END_VAR
	VAR
		intern : Motorky_Intern_typ;
		internFI : Motorky_InternFI_typ;
	END_VAR
END_FUNCTION_BLOCK

FUNCTION_BLOCK MM
	VAR_INPUT
		init : Motorky_Init_MM_typ;
		cmd : Motorky_Cmd_typ;
		param : Motorky_Param_typ;
	END_VAR
	VAR_OUTPUT
		info : Motorky_Info_typ;
		IOMapping : Motorky_MM_IOMapping;
	END_VAR
	VAR
		intern : Motorky_Intern_typ;
		internMM : Motorky_InternMM_typ;
	END_VAR
END_FUNCTION_BLOCK

FUNCTION_BLOCK DS
	VAR_INPUT
		init : Motorky_Init_NoEnc_typ;
		cmd : Motorky_Cmd_typ;
		param : Motorky_Param_typ;
	END_VAR
	VAR_OUTPUT
		info : Motorky_Info_typ;
		IOMapping : Motorky_DS_IOMapping;
	END_VAR
	VAR
		intern : Motorky_Intern_typ;
		movTargetTimeOffset : DINT;
		units2output : Motorky_ConvertPosition;
	END_VAR
END_FUNCTION_BLOCK

FUNCTION_BLOCK SM
	VAR_INPUT
		init : Motorky_Init_SM_typ;
		cmd : Motorky_Cmd_typ;
		param : Motorky_Param_typ;
	END_VAR
	VAR_OUTPUT
		info : Motorky_Info_typ;
		IOMapping : Motorky_SM_IOMapping;
	END_VAR
	VAR
		intern : Motorky_Intern_typ;
		tofBoostCurrent : Motorky_TOF;
		dPosition : DINT;
		oldPosition : DINT;
		units2output : Motorky_ConvertPosition;
		filterLevel : INT;
	END_VAR
END_FUNCTION_BLOCK
```

#### ds.c
```c
/***********************************************************************************************
	DEFINES
************************************************************************************************/
#define RESET_OUTPUT 	ConvertPositionInitialize(pUnits2output, p->init.units, p->init.microsteps, p->init.reverseDirection, pPathGenerator->outputPosition, pUnits2output->output);

/***********************************************************************************************
	INCLUDES
************************************************************************************************/
#include <motorky.h>
#include <string.h>
#include "path_generator.h"
#include "auxiliaries.h"

/****************************************************************************
Function    : DS()
Author      : RV
Description : Main function to control a stepper motor modul with a DS modul
Date        : 7.12.2006
Changes     :
****************************************************************************/
void DS(DS_typ *p)
{
	Motorky_DS_IOMapping		*pIOMapping = &p->IOMapping;
	Motorky_Intern_typ			*pIntern = &p->intern;
	Motorky_PathGenerator		*pPathGenerator = &pIntern->pathGenerator;
//	Motorky_ActualSpeed			*pActualSpeed = &pIntern->actualSpeed;
	Motorky_MoveActive 			*pMoveActive = &pIntern->moveActive;
	Motorky_ConvertPosition		*pUnits2output = &p->units2output;

/***********************************************************************************************
	CHECK ERRORS
************************************************************************************************/

	#include "check_errors.h"

/***********************************************************************************************
	BIG STATE MACHINE
************************************************************************************************/
	switch(pIntern->step)
	{
/***********************************************************************************************
	STATES 0 - 99 PERFORM INITIALIZATION
************************************************************************************************/
	case 0:
		p->movTargetTimeOffset = 4*ConvertTime(p->init.taskTime);

		pIntern->step = 10;
		break;

/***********************************************************************************************
	BASIC STATES 10 - 1009
************************************************************************************************/
	#include "basic.h"

	case 1010:
		p->info.status = 0;

		/*	return from error */
		if (p->info.initialized)
		{
			pIntern->step = 100;
		}
		else
		{
			pIntern->step = 0;
		}
		break;
	}

	#include "every_cycle.h"

/***********************************************************************************************
	OUTPUT GENERATOR
************************************************************************************************/
	ConvertPosition(pUnits2output,pPathGenerator->outputPosition);

	pIOMapping->MovTargetPosition = pUnits2output->output ;
	pIOMapping->MovTargetTime = pIOMapping->SystemTime + p->movTargetTimeOffset;
}
```

#### fi.c
```c
/***********************************************************************************************
	DEFINES
************************************************************************************************/
#define ENCODER_POSITION pIOMapping->Encoder
#define ENCODER_USED
#define RESET_OUTPUT

/***********************************************************************************************
	INCLUDES
************************************************************************************************/
#include <motorky.h>
#include <string.h>
#include "path_generator.h"
#include "auxiliaries.h"

/****************************************************************************
Function    : FI()
Author      : RV
Description : Main function to control a frequency invertor with signal +-10V
Date        : 5.2.2008
Changes     :
****************************************************************************/
void FI(FI_typ *p)
{
	Motorky_FI_IOMapping			*pIOMapping = &p->IOMapping;
	Motorky_Intern_typ				*pIntern = &p->intern;
	Motorky_InternFI_typ			*pInternFI = &p->internFI;
	Motorky_PathGenerator			*pPathGenerator = &pIntern->pathGenerator;
	Motorky_ActualSpeed				*pActualSpeed = &pInternFI->actualSpeed;
	Motorky_MoveActive 				*pMoveActive = &pIntern->moveActive;
	Motorky_ConvertPosition			*pEncoder2units = &pInternFI->encoder2units;
	Motorky_PID						*pPID = &pInternFI->pid;

/***********************************************************************************************
	CHECK ERRORS
************************************************************************************************/
	#include "check_errors.h"

/***********************************************************************************************
	BIG STATE MACHINE
************************************************************************************************/
	switch(pIntern->step)
	{
/***********************************************************************************************
	STATES 0 - 99 PERFORM INITIALIZATION
************************************************************************************************/
	case 0:
		pIntern->step = 10;
		break;

/***********************************************************************************************
	BASIC STATES 10 - 1009
************************************************************************************************/
	#include "basic.h"

	case 1010:
		p->info.status = 0;

		/*	return from error */
		if (p->info.initialized)
		{
			pIntern->step = 100;
		}
		else
		{
			pIntern->step = 0;
		}
		break;
	}

	#include "every_cycle.h"

/***********************************************************************************************
	OUTPUT GENERATOR
************************************************************************************************/
	pPID->enable =  p->info.powerOn;
	pPID->W = pPathGenerator->outputPosition;
	pPID->X = pEncoder2units->output;
	PID(pPID);
	if (pEncoder2units->reverseDirection)
	{
		pIOMapping->AnalogOutput = -pPID->Y;
	}
	else
	{
		pIOMapping->AnalogOutput = pPID->Y;
	}
}
```

#### mm.c
```c
/***********************************************************************************************
	DEFINES
************************************************************************************************/
#define ENCODER_POSITION pIOMapping->Counter
#define ENCODER_USED
#define RESET_OUTPUT
#define SPEED_PID_USED

/***********************************************************************************************
	INCLUDES
************************************************************************************************/
#include <motorky.h>
#include <string.h>
#include "path_generator.h"
#include "auxiliaries.h"

/****************************************************************************
Function    : MM()
Author      : RV
Description : Main function to control a MM motor modul
Date        : 5.2.2008
Changes     :
****************************************************************************/
void MM(MM_typ *p)
{
	Motorky_MM_IOMapping			*pIOMapping = &p->IOMapping;
	Motorky_Intern_typ				*pIntern = &p->intern;
	Motorky_InternMM_typ			*pInternMM = &p->internMM;
	Motorky_PathGenerator			*pPathGenerator = &pIntern->pathGenerator;
	Motorky_ActualSpeed				*pActualSpeed = &pInternMM->actualSpeed;
	Motorky_MoveActive 				*pMoveActive = &pIntern->moveActive;
	Motorky_ConvertPosition			*pEncoder2units = &pInternMM->encoder2units;
	Motorky_PID						*pPID = &pInternMM->pid;
	Motorky_PID						*pSpeedPID = &pInternMM->speedPID;

/***********************************************************************************************
	CHECK ERRORS
************************************************************************************************/
	if (pIOMapping->UnderVoltageError)
	{
		p->info.status = ERR_UNDER_VOLTAGE;
	}

	if (pIOMapping->OverVoltageError)
	{
		p->info.status = ERR_OVER_VOLTAGE;
	}

	if (pIOMapping->OvertemperatureError)
	{
		p->info.status = ERR_OVER_TEMPERATURE;
	}

	if (pIOMapping->OvercurrentError)
	{
		p->info.status = ERR_OVER_CURRENT;
	}

	#include "check_errors.h"

/***********************************************************************************************
	BIG STATE MACHINE
************************************************************************************************/
	switch(pIntern->step)
	{
/***********************************************************************************************
	STATES 0 - 99 PERFORM INITIALIZATION
************************************************************************************************/
	case 0:
		pIOMapping->PeriodDuration = 50;/* 100 us ... 10 kHz */
		pIntern->step = 10;
		break;

/***********************************************************************************************
	BASIC STATES 10 - 1009
************************************************************************************************/
	#include "basic.h"

	case 1010:
		/*	acknowledge motor error */
		pIOMapping->ClearError = 1;
		pIntern->step++;
		break;

	case 1011:
		/*	acknowledge motor error */
		pIOMapping->ClearError = 0;
		pIntern->step++;
		break;

	case 1012:
		p->info.status = 0;

		/*	return from error */
		if (p->info.initialized)
		{
			pIntern->step = 100;
		}
		else
		{
			pIntern->step = 0;
		}
		break;
	}

	#include "every_cycle.h"

/***********************************************************************************************
	OUTPUT GENERATOR
************************************************************************************************/
	/*	position PID */
	pPID->enable =  p->info.powerOn;
	pPID->W = pPathGenerator->outputPosition;
	pPID->X = pEncoder2units->output;
	PID(pPID);

	/* speed PID */
	pSpeedPID->enable =  p->info.powerOn;
	pSpeedPID->W = pPID->Y;
	pSpeedPID->X = pActualSpeed->actSpeed;
	PID(pSpeedPID);

	pIOMapping->PulseWidth = pSpeedPID->Y;

	if (pEncoder2units->reverseDirection)
	{
		pIOMapping->PulseWidth = -pIOMapping->PulseWidth;
	}
}
```

#### sm.c
```c
/***********************************************************************************************
	DEFINES
************************************************************************************************/
#define RESET_OUTPUT 	ConvertPositionInitialize(pUnits2output, p->init.units, p->init.microsteps, p->init.reverseDirection, \
						pPathGenerator->outputPosition, pUnits2output->output);

/***********************************************************************************************
	INCLUDES
************************************************************************************************/
#include <motorky.h>
#include <string.h>
#include "path_generator.h"
#include "auxiliaries.h"

/****************************************************************************
Function    : SM()
Author      : RV
Description : Main function to control a stepper motor modul
Date        : 7.12.2006
Changes     :
****************************************************************************/
void SM(SM_typ *p)
{
	Motorky_SM_IOMapping		*pIOMapping = &p->IOMapping;
	Motorky_Intern_typ			*pIntern = &p->intern;
	Motorky_PathGenerator		*pPathGenerator = &pIntern->pathGenerator;
	Motorky_MoveActive 			*pMoveActive = &pIntern->moveActive;
	Motorky_ConvertPosition		*pUnits2output = &p->units2output;

/***********************************************************************************************
	CHECK ERRORS
************************************************************************************************/
	if (pIOMapping->StallError)
	{
		p->info.status = ERR_STALL;
	}

	if (pIOMapping->OvertemperatureError)
	{
		p->info.status = ERR_OVER_TEMPERATURE;
	}

	if (pIOMapping->OvercurrentError)
	{
		p->info.status = ERR_OVER_CURRENT;
	}

	if (pIOMapping->ModulePowerSupplyError)
	{
		p->info.status = ERR_POWER_SUPPLY_ERROR;
	}

	if (pIOMapping->UZKStatus == 0)
	{
		p->info.status = ERR_LOW_DC_BUS_VOLTAGE;
	}

//	if (pIOMapping->Enable == 0)
//	{
//		p->info.status = ERR_ENABLE_INPUT_NOT_ACTIVE;
//	}
	#include "check_errors.h"

/***********************************************************************************************
	BIG STATE MACHINE
************************************************************************************************/
	switch(pIntern->step)
	{
/***********************************************************************************************
	STATES 0 - 99 PERFORM INITIALIZATION
************************************************************************************************/
	case 0:

		TOFInitialize(&p->tofBoostCurrent,p->init.taskTime, 0.1); // =100ms

		if (p->init.outputFilter < 0) p->init.outputFilter = 0;
		if (p->init.outputFilter > 0.1) p->init.outputFilter = 0.1;

		if (p->init.taskTime > 0)
		{
			p->filterLevel = 1 + p->init.outputFilter / p->init.taskTime;
		}

		pIntern->step = 10;
		break;

/***********************************************************************************************
	BASIC STATES 10 - 1009
************************************************************************************************/
	#include "basic.h"

	case 1010:
		/*	acknowledge motor error */
		pIOMapping->ClearError = 1;
		pIntern->step++;
		break;

	case 1011:
		/*	acknowledge motor error */
		pIOMapping->ClearError = 0;
		pIntern->step++;
		break;

	case 1012:
		/*	wait till module resets error */
		pIntern->step++;
		break;

	case 1013:
		p->info.status = 0;
		/*	return from error */
		if (p->info.initialized)
		{
			pIntern->step = 100;
		}
		else
		{
			pIntern->step = 0;
		}
		break;
	}

	#include "every_cycle.h"

/***********************************************************************************************
	OUTPUT GENERATOR
************************************************************************************************/
	ConvertPosition(pUnits2output,pPathGenerator->outputPosition);

	pIOMapping->DriveEnable = p->info.powerOn;

	p->dPosition  = pUnits2output->output - p->oldPosition;

	pIOMapping->MotorStep0 = 0;

	if (p->dPosition > 0)
	{
		if (p->dPosition >= p->filterLevel)
		{
			pIOMapping->MotorStep0 = p->dPosition / p->filterLevel;
		}
		else
		{
			pIOMapping->MotorStep0 = 1;
		}
	}

	if (p->dPosition < 0)
	{
		if (p->dPosition <= -p->filterLevel)
		{
			pIOMapping->MotorStep0 = p->dPosition / p->filterLevel;
		}
		else
		{
			pIOMapping->MotorStep0 = -1;
		}
	}

	p->oldPosition += pIOMapping->MotorStep0;

	/*	determine if boost current should be used */
	if 	(pPathGenerator->motionState == MOTION_STATE_ACCELERATING || pPathGenerator->motionState == MOTION_STATE_DECELERATING)
	{
		p->tofBoostCurrent.IN = 1;
	}
	else
	{
		p->tofBoostCurrent.IN = 0;
	}

	TOF(&p->tofBoostCurrent);
	pIOMapping->BoostCurrent = p->tofBoostCurrent.Q;

	if (pPathGenerator->motionState == MOTION_STATE_STANDSTILL && p->tofBoostCurrent.Q == 0)
	{
		pIOMapping->StandstillCurrent = 1;
	}
	else
	{
		pIOMapping->StandstillCurrent = 0;
	}

}
```

#### path_generator.h
```c
/********************************************************************
 * COPYRIGHT --
 ********************************************************************
 * Library: Motorky
 * File: path_generator.h
 * Author: vancurar
 * Created: June 29, 2008
 *******************************************************************/

#include <bur/plctypes.h>

void PathGenerator(Motorky_PathGenerator *pPathGenerator);

void PathGeneratorInitialize(Motorky_PathGenerator *pPathGenerator, REAL taskTime);

void PathGeneratorResetError(Motorky_PathGenerator *pPathGenerator);

void PathGeneratorSetPosition(Motorky_PathGenerator *pPathGenerator, DINT position);

#define ABS(c)		(((c) >= 0) ? (c) : -(c))
```

#### path_generator.c
```c
#include <motorky.h>
#include "auxiliaries.h"
#include "speed_ramping.h"

/*	this function determines pPathGenerator->vn and pPathGenerator->sn */
void PathGenerator(Motorky_PathGenerator *pPathGenerator)
{
	Motorky_SpeedRamping *pSpeedRamping = &pPathGenerator->speedRamping;
	DINT	distance, distance2;
	DINT	requiredDeceleration;

	/*	decide if SW limits are used */
	if (pPathGenerator->positiveSwLimit > pPathGenerator->negativeSwLimit)
	{
		/*	if going in positive direction */
		if (pPathGenerator->outputSpeed > 0)
		{
			/*	compute distance to SW limit */
			distance = pPathGenerator->positiveSwLimit - pPathGenerator->outputPosition;

			/*	compute required deceleration ramp */
			if (distance != 0)
			{
				requiredDeceleration = ABS(((long long)pPathGenerator->outputSpeed*pPathGenerator->outputSpeed)/(2*distance));
			}
			else
			{
				requiredDeceleration = 0;
			}

			if (distance < 0 || (distance > 0 && requiredDeceleration >= pPathGenerator->deceleration))
			{
				/*	set error */
				pPathGenerator->status = ERR_POSITIVE_SW_LIMIT_REACHED;

				pPathGenerator->moveCommand = MOVE_COMMAND_STOP;
			}
		}
		/*	if going in negative direction */
		else if (pPathGenerator->outputSpeed < 0)
		{
			/*	compute distance to SW limit */
			distance = pPathGenerator->negativeSwLimit - pPathGenerator->outputPosition;

			/*	compute required deceleration ramp */
			if (distance != 0)
			{
				requiredDeceleration = ABS(((long long)pPathGenerator->outputSpeed*pPathGenerator->outputSpeed)/(2*distance));
			}
			else
			{
				requiredDeceleration = 0;
			}

			if (distance > 0 || (distance < 0 && requiredDeceleration >= pPathGenerator->deceleration))
			{
				/*	set error */
				pPathGenerator->status = ERR_NEGATIVE_SW_LIMIT_REACHED;

				pPathGenerator->moveCommand = MOVE_COMMAND_STOP;
			}
		}
	}

	/* MOVE_ABSOLUTE */
	if (pPathGenerator->moveCommand == MOVE_COMMAND_ABSOLUTE)
	{
		/*	distance to go */
		distance = pPathGenerator->setPosition - pPathGenerator->outputPosition;

		/*	compute required deceleration ramp */
		if (distance != 0)
		{
			requiredDeceleration = ABS(((long long)pPathGenerator->outputSpeed*pPathGenerator->outputSpeed)/(2*distance));
		}
		else
		{
			requiredDeceleration = 0;
		}

		/*	must decelerate? */
		if (requiredDeceleration >= pPathGenerator->deceleration)
		{
			pSpeedRamping->setSpeed = 0;
			pSpeedRamping->acceleration = pPathGenerator->acceleration;
			pSpeedRamping->deceleration = requiredDeceleration;
		}
		else
		{
			/*	compute speed */
			if (distance > 0)
			{
				/*	go in positive direction */
				pSpeedRamping->setSpeed = ABS(pPathGenerator->setSpeed);
				pSpeedRamping->acceleration = pPathGenerator->acceleration;
				pSpeedRamping->deceleration = pPathGenerator->deceleration;
			}
			else if (distance < 0)
			{
				/*	go in negative direction */
				pSpeedRamping->setSpeed = -ABS(pPathGenerator->setSpeed);
				pSpeedRamping->acceleration = pPathGenerator->acceleration;
				pSpeedRamping->deceleration = pPathGenerator->deceleration;
			}
			else
			{
				/*	stop movement */
				pSpeedRamping->setSpeed = 0;
				pSpeedRamping->acceleration = pPathGenerator->acceleration;
				pSpeedRamping->deceleration = pPathGenerator->deceleration;
			}
		}

		/*	call speed ramping FUB */
		SpeedRamping(pSpeedRamping);

		/*	distance to go */
		distance2 = pPathGenerator->setPosition - pSpeedRamping->actualPosition;

		/*	detect if target position was reached */
		if ((distance > 0 && distance2 <= 0) || (distance < 0 && distance2 >=0))
		{
			SpeedRampingSetPosition(pSpeedRamping, pPathGenerator->setPosition);
			SpeedRampingSetSpeed(pSpeedRamping, 0);
		}
	}
	/* MOVE_VELOCITY */
	else if (pPathGenerator->moveCommand == MOVE_COMMAND_VELOCITY)
	{
		pSpeedRamping->setSpeed = pPathGenerator->setSpeed;
		pSpeedRamping->acceleration = pPathGenerator->acceleration;
		pSpeedRamping->deceleration = pPathGenerator->deceleration;

		/*	call speed ramping FUB */
		SpeedRamping(pSpeedRamping);
	}
	/* MOVE_STOP */
	else if (pPathGenerator->moveCommand == MOVE_COMMAND_STOP)
	{
		/*	must decelerate */
		pSpeedRamping->setSpeed = 0;
		pSpeedRamping->acceleration = pPathGenerator->acceleration;
		pSpeedRamping->deceleration = pPathGenerator->deceleration;

		/*	call speed ramping FUB */
		SpeedRamping(pSpeedRamping);
	}

	/*	copy actual position and speed */
	pPathGenerator->outputPosition = pSpeedRamping->actualPosition;
	pPathGenerator->outputSpeed = pSpeedRamping->actualSpeed;

	/*	copy motion state */
	if (pSpeedRamping->motionState == MOTION_STATE_CONSTANT_SPEED && pSpeedRamping->actualSpeed == 0)
	{
		/*	MOTION_STATE_STANDSTILL is a special case of MOTION_STATE_CONSTANT_SPEED */
		pPathGenerator->motionState = MOTION_STATE_STANDSTILL;
	}
	else
	{
		pPathGenerator->motionState = pSpeedRamping->motionState;
	}
}

/*	This function initializes PathGenerator */
void PathGeneratorInitialize(Motorky_PathGenerator *pPathGenerator, REAL taskTime)
{
	SpeedRampingInitialize(&pPathGenerator->speedRamping, ConvertTime(taskTime));
}

/*	This function resets error in PathGenerator */
void PathGeneratorResetError(Motorky_PathGenerator *pPathGenerator)
{
	pPathGenerator->status = 0;
}

/*	This function sets internal position to desired value */
void PathGeneratorSetPosition(Motorky_PathGenerator *pPathGenerator, DINT position)
{
	pPathGenerator->setPosition = position;
	SpeedRampingSetPosition(&pPathGenerator->speedRamping, position);
	pPathGenerator->outputPosition = position;
}
```

#### speed_ramping.h
```c
/********************************************************************
 * COPYRIGHT --
 ********************************************************************
 * Library: Motorky
 * File: speed_ramping.h
 * Author: vancurar
 * Created: June 29, 2008
 *******************************************************************/

#include <bur/plctypes.h>

void SpeedRamping(Motorky_SpeedRamping *pSpeedRamping);

void SpeedRampingInitialize(Motorky_SpeedRamping *pSpeedRamping, DINT taskTime);

void SpeedRampingSetPosition(Motorky_SpeedRamping *pSpeedRamping, DINT position);

void SpeedRampingSetSpeed(Motorky_SpeedRamping *pSpeedRamping, DINT speed);

#define ABS(c)		(((c) >= 0) ? (c) : -(c))
```

#### speed_ramping.c
```c
#include <motorky.h>
#include "speed_ramping.h"

/*	compute new speed and position */
void SpeedRamping(Motorky_SpeedRamping *pSpeedRamping)
{
	DINT speedDifference;
	DINT absoluteSpeedDifference;
	DINT speedDifference2;

	/*	compute speed difference */
	speedDifference = pSpeedRamping->setSpeed - pSpeedRamping->actualSpeed;

	if (speedDifference > 0)
	{
		/*	compute absolute speed difference */
		absoluteSpeedDifference = ABS(pSpeedRamping->setSpeed) - ABS(pSpeedRamping->actualSpeed);

		/*	speed must be increased ? */
		if (absoluteSpeedDifference > 0)
		{
			/*	accelerate in positive direction  */
			pSpeedRamping->vIntegral += pSpeedRamping->acceleration;
			/*	set state "accelerating" */
			pSpeedRamping->motionState = MOTION_STATE_ACCELERATING;
		}
		else
		{
			/*	decelerate in positive direction */
			pSpeedRamping->vIntegral += pSpeedRamping->deceleration;
			/*	set state "decelerating" */
			pSpeedRamping->motionState = MOTION_STATE_DECELERATING;
		}
	}
	else if (speedDifference < 0)
	{
		/*	compute absolute speed difference */
		absoluteSpeedDifference = ABS(pSpeedRamping->setSpeed) - ABS(pSpeedRamping->actualSpeed);

		/*	speed must be increased ? */
		if (absoluteSpeedDifference > 0)
		{
			/*	accelerate in negative direction */
			pSpeedRamping->vIntegral -= pSpeedRamping->acceleration;
			/*	set state "accelerating" */
			pSpeedRamping->motionState = MOTION_STATE_ACCELERATING;
		}
		else
		{
			/*	decelerate in negative direction */
			pSpeedRamping->vIntegral -= pSpeedRamping->deceleration;
			/*	set state "decelerating" */
			pSpeedRamping->motionState = MOTION_STATE_DECELERATING;
		}
	}
	else
	{
		/*	no speed change is needed */
		pSpeedRamping->motionState = MOTION_STATE_CONSTANT_SPEED;
	}

	/*	compute new value of speed */
	pSpeedRamping->actualSpeed += pSpeedRamping->vIntegral/pSpeedRamping->divisor;
	pSpeedRamping->vIntegral %= pSpeedRamping->divisor;

	/*	check if speed was not reached */
	speedDifference2 = pSpeedRamping->setSpeed - pSpeedRamping->actualSpeed;

	if ((speedDifference > 0 && speedDifference2 <= 0)||(speedDifference < 0 && speedDifference2 >= 0))
	{
		pSpeedRamping->actualSpeed = pSpeedRamping->setSpeed;
		pSpeedRamping->vIntegral = 0;
		pSpeedRamping->motionState = MOTION_STATE_CONSTANT_SPEED;
	}

	/*	compute new position */
	pSpeedRamping->sIntegral += pSpeedRamping->actualSpeed;
	pSpeedRamping->actualPosition += pSpeedRamping->sIntegral/pSpeedRamping->divisor;
	pSpeedRamping->sIntegral %= pSpeedRamping->divisor;
}

void SpeedRampingSetPosition(Motorky_SpeedRamping *pSpeedRamping, DINT position)
{
	pSpeedRamping->actualPosition = position;
	pSpeedRamping->sIntegral = 0;
}

void SpeedRampingSetSpeed(Motorky_SpeedRamping *pSpeedRamping, DINT speed)
{
	pSpeedRamping->actualSpeed = speed;
	pSpeedRamping->vIntegral = 0;
}

void SpeedRampingInitialize(Motorky_SpeedRamping *pSpeedRamping, DINT taskTime)
{
	/*	compute divisor */
	pSpeedRamping->divisor = 1000000/taskTime;
}
```

#### check_errors.h
```c
	if (/*pIntern->step >= 100 && */pIntern->step < 1000)
	{
		/* check if drive is ready */
		if (p->info.powerOn && pIOMapping->DriveReady == 0)
		{
			p->info.status = ERR_DRIVE_NOT_READY;
		}

		#ifdef ENCODER_POSITION
			/*	check lag error */
			if (p->info.powerOn && ABS(p->info.lagError) > p->init.maxLagError)
			{
				p->info.status = ERR_LAG_ERROR;
			}
		#endif

		/*	check limit switches, but not in homing steps */
		if(pIntern->step < 200 || pIntern->step >= 300)
		{
			/*	if negative limit switch is closed */
			if (p->IOMapping.negativeLimitSwitch == 1)
			{
				/*	and we go in negative direction */
				if (pPathGenerator->outputSpeed < 0)
				{
					p->info.status = ERR_NEGATIVE_LIMIT_SWITCH_CLOSED;
				}
			}

			/*	if positive switch is closed */
			if (p->IOMapping.positiveLimitSwitch == 1)
			{
				/*	and we go in positive direction */
				if (pPathGenerator->outputSpeed > 0)
				{
					p->info.status = ERR_POSITIVE_LIMIT_SWITCH_CLOSED;
				}
			}
		}

		/*	check error from path generator */
		if (pPathGenerator->status == ERR_POSITIVE_SW_LIMIT_REACHED && pPathGenerator->motionState == MOTION_STATE_STANDSTILL)
		{
			p->info.status = ERR_POSITIVE_SW_LIMIT_REACHED;
		}

		if (pPathGenerator->status == ERR_NEGATIVE_SW_LIMIT_REACHED && pPathGenerator->motionState == MOTION_STATE_STANDSTILL)
		{
			p->info.status = ERR_NEGATIVE_SW_LIMIT_REACHED;
		}

		if 	(p->info.status != 0)
		{
			/*	new error */
			pIntern->oldStep = pIntern->step;
			/*	go to error step */
			pIntern->step = 1000;
		}
		else
		{
			/*	acknowledge pressed and there is no error, reset request */
			if (p->cmd.acknowledge)
			{
				p->cmd.acknowledge = 0;
			}

			/*	stop pressed? */
			if (p->cmd.stop == 1 || p->cmd.power == 0)
			{
				/*	if moving, go to stop step */
				if (pPathGenerator->motionState != MOTION_STATE_STANDSTILL)
				{
					pIntern->step = 180;
				}

				/*	clear all commands, except of cmd.power */
				if (p->cmd.stop == 1) p->cmd.homing = 0;
				p->cmd.absolute = 0;
				p->cmd.additive = 0;
				p->cmd.cyclicPosition = 0;
				p->cmd.velocity = 0;
				p->cmd.acknowledge = 0;
				p->cmd.stop = 0;
			}
		}
	}
```

#### basic.h
```c
/***********************************************************************************************
	INITIALIZATION STATE
***********************************************************************************************/
case 10:
		/*	default initialization */
		if (p->init.units < 1) p->init.units = 1;

		if (p->init.taskTime <= 0 || p->init.taskTime >= 1)
		{
			p->info.status = ERR_WRONG_TASK_TIME;
			return;
		}

		if (p->init.settleTime == 0) p->init.settleTime = 0;

		if (p->param.position == 0) p->param.position = 1000;
		if (p->param.speed == 0) p->param.speed = DEFAULT_SPEED;
		if (p->param.acceleration == 0) p->param.acceleration = DEFAULT_ACCELERATION;
		if (p->param.deceleration == 0) p->param.deceleration = DEFAULT_ACCELERATION;

		if (p->param.homing.speed2 == 0) p->param.homing.speed2 = p->param.speed;

		/*	initialize path generator */
		PathGeneratorInitialize(pPathGenerator, p->init.taskTime);

		#ifdef ENCODER_USED
			/*	default initialization */
			if (p->init.maxLagError == 0) p->init.maxLagError = 1000;
			if (p->init.Kp == 0) p->init.Kp = 1;
			/*if (p->init.Tn == 0) p->init.Tn = 0;*/

			if (p->init.encoderIncrements == 0)
			{
				p->info.status = ERR_WRONG_ENCODER_INCREMENTS;
				return;
			}
			/*	initialize conversion */
			ConvertPositionInitialize(pEncoder2units,p->init.encoderIncrements,p->init.units,p->init.reverseDirection,
				ENCODER_POSITION,p->info.position);

			ActualSpeedInitialize(pActualSpeed, p->init.taskTime, p->init.speedFilter);

		#else
			if (p->init.microsteps == 0) p->init.microsteps = 200*256;
		#endif

		#ifdef SPEED_PID_USED
			if (p->init.speedKp == 0) p->init.speedKp = 0.01;
			/*if (p->init.speedTn == 0) p->init.speedTn = 0;*/
		#endif

		MoveActiveInitialize(pMoveActive, p->init.taskTime, p->init.settleTime);

		RESET_OUTPUT

		p->info.initialized = 1;
		pIntern->step = 100;

/***********************************************************************************************
	COMMAND STATE
***********************************************************************************************/
	case 100:
		if (p->cmd.power && !p->info.powerOn)
		{
			/*	switch power on */
			pIntern->step = 110;
		}

		if (!p->cmd.power && p->info.powerOn)
		{
			/*	switch power off */
			pIntern->step = 120;
		}

		if (p->cmd.homing)
		{
			pIntern->step = 200;
			goto L_200;
		}

		if (p->cmd.absolute)
		{
			pIntern->step = 140;
			goto L_140;
		}

		if (p->cmd.additive)
		{
			pIntern->step = 150;
			goto L_150;
		}

		if (p->cmd.cyclicPosition)
		{
			pIntern->step = 160;
			goto L_160;
		}

		if (p->cmd.velocity)
		{
			pIntern->step = 170;
			goto L_170;
		}
		break;

/***********************************************************************************************
	SWITCH CONTROLLER ON
***********************************************************************************************/
	case 110:
		/*	switch on output */
		p->info.powerOn = 1;

		/*	set intern position inside path generator to actual position */
		PathGeneratorSetPosition(pPathGenerator, p->info.position);

		#ifdef ENCODER_USED
			/*	intialize speed filter */
			ActualSpeedInitialize(pActualSpeed, p->init.taskTime, p->init.speedFilter);

			/*	initialize PID */
			#ifdef SPEED_PID_USED
				PIDInitialize(pPID, p->init.Kp, p->init.Tn, p->init.taskTime, DINT_MAXVALUE, -DINT_MAXVALUE);
				PIDInitialize(pSpeedPID, p->init.speedKp, p->init.speedTn, p->init.taskTime, INT_MAXVALUE, -INT_MAXVALUE);
			#else
				PIDInitialize(pPID, p->init.Kp, p->init.Tn, p->init.taskTime, INT_MAXVALUE, -INT_MAXVALUE);
			#endif
		#endif

		pIntern->step = 100;
		break;

/***********************************************************************************************
	SWITCH CONTROLLER OFF
************************************************************************************************/
	case 120:

		p->info.powerOn = 0;
		pIntern->step = 100;
		break;

/***********************************************************************************************
	ABSOLUTE MOVE
************************************************************************************************/
	case 140:
L_140:
		/*	prepare data for path generator */
		pPathGenerator->moveCommand = MOVE_COMMAND_ABSOLUTE;
		pPathGenerator->setPosition = p->param.position;
		pPathGenerator->setSpeed = p->param.speed;
		pPathGenerator->acceleration = p->param.acceleration;
		pPathGenerator->deceleration = p->param.deceleration;
		pPathGenerator->positiveSwLimit = p->init.positiveSwLimit;
		pPathGenerator->negativeSwLimit = p->init.negativeSwLimit;

		/*	clear flag */
		p->cmd.absolute = 0;
		pIntern->step = 100;
		break;

/***********************************************************************************************
	ADDITIVE MOVE
************************************************************************************************/
	case 150:
L_150:
		/*	prepare data for path generator */
		pPathGenerator->moveCommand = MOVE_COMMAND_ABSOLUTE;
		pPathGenerator->setPosition = pPathGenerator->outputPosition + p->param.position;
		pPathGenerator->setSpeed = p->param.speed;
		pPathGenerator->acceleration = p->param.acceleration;
		pPathGenerator->deceleration = p->param.deceleration;
		pPathGenerator->positiveSwLimit = p->init.positiveSwLimit;
		pPathGenerator->negativeSwLimit = p->init.negativeSwLimit;

		/*	clear flag */
		p->cmd.additive = 0;
		pIntern->step = 100;
		break;

/***********************************************************************************************
	POSITION MOVEMENT
************************************************************************************************/
	case 160:
L_160:
		pPathGenerator->moveCommand = MOVE_COMMAND_ABSOLUTE;
		pPathGenerator->setPosition = p->param.position;
		pPathGenerator->setSpeed = p->param.speed;
		pPathGenerator->acceleration = p->param.acceleration;
		pPathGenerator->deceleration = p->param.deceleration;
		pPathGenerator->positiveSwLimit = p->init.positiveSwLimit;
		pPathGenerator->negativeSwLimit = p->init.negativeSwLimit;

		/*	attempt to stop? */
		if (p->cmd.cyclicPosition == 0)
		{
			pPathGenerator->moveCommand = MOVE_COMMAND_STOP;
			pIntern->step=100;
		}
		break;

/***********************************************************************************************
	VELOCITY MOVEMENT
************************************************************************************************/
	case 170:
L_170:
		pPathGenerator->moveCommand = MOVE_COMMAND_VELOCITY;
		pPathGenerator->setSpeed = p->param.speed;
		pPathGenerator->acceleration = p->param.acceleration;
		pPathGenerator->deceleration = p->param.deceleration;
		pPathGenerator->positiveSwLimit = p->init.positiveSwLimit;
		pPathGenerator->negativeSwLimit = p->init.negativeSwLimit;

		/*	attempt to stop? */
		if (p->cmd.velocity == 0)
		{
			pPathGenerator->moveCommand = MOVE_COMMAND_STOP;
			pIntern->step = 100;
		}
		break;

/***********************************************************************************************
	STOP MOVEMENT
************************************************************************************************/
	case 180:
		pPathGenerator->moveCommand = MOVE_COMMAND_STOP;
		pPathGenerator->deceleration = p->param.deceleration;

		/*	wait till movement stopped */
		if (pPathGenerator->motionState == MOTION_STATE_STANDSTILL)
		{
			pIntern->step=100;
		}
		break;

/***********************************************************************************************
	HOMING STATES
************************************************************************************************/
	case 200:
L_200:
		/*	reset flag */
		p->info.homingOk = 0;

		/*	set acceleration and deceleration */
		pPathGenerator->acceleration = p->param.acceleration;
		pPathGenerator->deceleration = p->param.deceleration;

		/*	set SW limits */
		pPathGenerator->positiveSwLimit = 0;
		pPathGenerator->negativeSwLimit = 0;

		/*	which homing mode */
		if (p->param.homing.mode == HOMING_DIRECT)
		{
			pIntern->step = 260;
		}
		else if (p->param.homing.mode == HOMING_END_SWITCH)
		{
			pIntern->step = 220;
		}
		else if (p->param.homing.mode == HOMING_REF_SWITCH)
		{
			pIntern->step = 240;
		}
		break;

/***********************************************************************************************
	HOMING_END_SWITCH
************************************************************************************************/
	case 220:

		/*	fast movement off positive HW end */
		if (p->IOMapping.positiveLimitSwitch)
		{
			pPathGenerator->moveCommand = MOVE_COMMAND_VELOCITY;
			pPathGenerator->setSpeed = -ABS(p->param.speed);
			break;
		}

		/*	fast movement off negative HW end */
		if (p->IOMapping.negativeLimitSwitch)
		{
			pPathGenerator->moveCommand = MOVE_COMMAND_VELOCITY;
			pPathGenerator->setSpeed = ABS(p->param.speed);
			break;
		}

		/*	fast movement to positive HW end */
		if (p->param.homing.edgeSwitch == DIRECTION_POSITIVE)
		{
			pPathGenerator->moveCommand = MOVE_COMMAND_VELOCITY;
			pPathGenerator->setSpeed = ABS(p->param.speed);
			pIntern->step = 221;
			break;
		}

		/*	fast movement to negative HW end */
		if (p->param.homing.edgeSwitch == DIRECTION_NEGATIVE)
		{
			pPathGenerator->moveCommand = MOVE_COMMAND_VELOCITY;
			pPathGenerator->setSpeed = -ABS(p->param.speed);
			pIntern->step = 224;
			break;
		}
		break;

	case 221:

		/*	turn when positive limit switch reached */
		if (p->IOMapping.positiveLimitSwitch)
		{
			/*	slow movement out off positive HW end */
			pPathGenerator->moveCommand = MOVE_COMMAND_VELOCITY;
			pPathGenerator->setSpeed = -ABS(p->param.homing.speed2);
			pIntern->step++;
		}
		break;

	case 222:

		if (p->IOMapping.positiveLimitSwitch ==0)
		{
			if (p->param.homing.triggerDirection == DIRECTION_NEGATIVE)
			{
				/*	finished */
				pPathGenerator->moveCommand = MOVE_COMMAND_STOP;
				pPathGenerator->deceleration = p->param.deceleration;
				pIntern->step = 250;
			}
			else
			{
				/*	change direction */
				pPathGenerator->moveCommand = MOVE_COMMAND_VELOCITY;
				pPathGenerator->setSpeed = ABS(p->param.homing.speed2);
				pIntern->step++;
			}
		}
		break;

	case 223:

		if (p->IOMapping.positiveLimitSwitch == 1)
		{
			/*	finished */
			pPathGenerator->moveCommand = MOVE_COMMAND_STOP;
			pPathGenerator->deceleration = p->param.deceleration;
			pIntern->step = 250;
		}
		break;

	case 224:

		/*	turn when negative limit switch reached */
		if (p->IOMapping.negativeLimitSwitch)
		{
			/*	slow movement out off negative HW end */
			pPathGenerator->moveCommand = MOVE_COMMAND_VELOCITY;
			pPathGenerator->setSpeed = ABS(p->param.homing.speed2);
			pIntern->step++;
		}
		break;

	case 225:

		if (p->IOMapping.negativeLimitSwitch == 0)
		{
			if (p->param.homing.triggerDirection == DIRECTION_POSITIVE)
			{
				/*	finished */
				pPathGenerator->moveCommand = MOVE_COMMAND_STOP;
				pPathGenerator->deceleration = p->param.deceleration;
				pIntern->step = 250;
			}
			else
			{
				/*	change direction */
				pPathGenerator->moveCommand = MOVE_COMMAND_VELOCITY;
				pPathGenerator->setSpeed = -ABS(p->param.homing.speed2);
				pIntern->step++;
			}
		}
		break;

	case 226:

		if (p->IOMapping.negativeLimitSwitch == 1)
		{
			/*	finished */
			pPathGenerator->moveCommand = MOVE_COMMAND_STOP;
			pPathGenerator->deceleration = p->param.deceleration;
			pIntern->step = 250;
		}
		break;

/***********************************************************************************************
	HOMING_REF_SWITCH
************************************************************************************************/
	case 240:

		/*	go with high speed in startDirection */
		if (p->param.homing.startDirection == DIRECTION_POSITIVE)
		{
			pPathGenerator->moveCommand = MOVE_COMMAND_VELOCITY;
			pPathGenerator->setSpeed = ABS(p->param.speed);
		}
		else
		{
			pPathGenerator->moveCommand = MOVE_COMMAND_VELOCITY;
			pPathGenerator->setSpeed = -ABS(p->param.speed);
		}
		pIntern->step++;
		break;

	case 241:

		/*	if right limit switch reached, turn direction */
		if (p->IOMapping.positiveLimitSwitch == 1)
		{
			pPathGenerator->moveCommand = MOVE_COMMAND_VELOCITY;
			pPathGenerator->setSpeed = -ABS(p->param.speed);
		}

		/*	if left limit switch reached, turn direction */
		if (p->IOMapping.negativeLimitSwitch == 1)
		{
			pPathGenerator->moveCommand = MOVE_COMMAND_VELOCITY;
			pPathGenerator->setSpeed = ABS(p->param.speed);
		}

		/*	detect positive edge of reference switch */
		if (p->IOMapping.referenceSwitch == 1 && pIntern->oldReferenceSwitch == 0)
		{
			/*	detect positive edge */
			if (pPathGenerator->outputSpeed > 0 && p->param.homing.edgeSwitch == DIRECTION_POSITIVE)
			{
				/*	slow down */
				pPathGenerator->moveCommand = MOVE_COMMAND_VELOCITY;
				pPathGenerator->setSpeed = -ABS(p->param.homing.speed2);
				pIntern->step++;
			}

			/*	detect negative edge */
			if (pPathGenerator->outputSpeed < 0 && p->param.homing.edgeSwitch == DIRECTION_NEGATIVE)
			{
				pPathGenerator->moveCommand = MOVE_COMMAND_VELOCITY;
				pPathGenerator->setSpeed = ABS(p->param.homing.speed2);
				pIntern->step++;
			}
		}

		/*	detect negative edge of reference switch */
		if (p->IOMapping.referenceSwitch == 0 && pIntern->oldReferenceSwitch == 1)
		{
			/*	detect negative edge */
			if (pPathGenerator->outputSpeed < 0)
			{
				if (p->param.homing.edgeSwitch == DIRECTION_POSITIVE)
				{
					pPathGenerator->moveCommand = MOVE_COMMAND_VELOCITY;
					pPathGenerator->setSpeed = ABS(p->param.homing.speed2);
					pIntern->step++;
				}
				else
				{
					/*	turn direction */
					pPathGenerator->moveCommand = MOVE_COMMAND_VELOCITY;
					pPathGenerator->setSpeed = ABS(p->param.speed);
				}
			}

			/*	detect positive edge */
			if (pPathGenerator->outputSpeed > 0)
			{
				if (p->param.homing.edgeSwitch == DIRECTION_NEGATIVE)
				{
					pPathGenerator->moveCommand = MOVE_COMMAND_VELOCITY;
					pPathGenerator->setSpeed = -ABS(p->param.homing.speed2);
					pIntern->step++;
				}
				else
				{
					/*	turn direction */
					pPathGenerator->moveCommand = MOVE_COMMAND_VELOCITY;
					pPathGenerator->setSpeed = -ABS(p->param.speed);
				}
			}
		}
		break;

	case 242:

		/*	detect positive edge of reference switch */
		if (p->IOMapping.referenceSwitch == 1 && pIntern->oldReferenceSwitch == 0)
		{
			if (pPathGenerator->outputSpeed > 0)
			{
				if (p->param.homing.triggerDirection == DIRECTION_POSITIVE)
				{
					/*	finished */
					pPathGenerator->moveCommand = MOVE_COMMAND_STOP;
					pPathGenerator->deceleration = p->param.deceleration;
					pIntern->step = 250;
				}
				else
				{
					/*	turn direction */
					pPathGenerator->moveCommand = MOVE_COMMAND_VELOCITY;
					pPathGenerator->setSpeed = -ABS(p->param.homing.speed2);
				}
			}

			if (pPathGenerator->outputSpeed < 0)
			{
				if (p->param.homing.triggerDirection == DIRECTION_NEGATIVE)
				{
					/*	finished */
					pPathGenerator->moveCommand = MOVE_COMMAND_STOP;
					pPathGenerator->deceleration = p->param.deceleration;
					pIntern->step = 250;
				}
				else
				{
					/*	turn direction */
					pPathGenerator->moveCommand = MOVE_COMMAND_VELOCITY;
					pPathGenerator->setSpeed = ABS(p->param.homing.speed2);
				}
			}
		}

		/*	detect negative edge of reference switch */
		if (p->IOMapping.referenceSwitch == 0 && pIntern->oldReferenceSwitch == 1)
		{
			if (pPathGenerator->outputSpeed > 0)
			{
				if (p->param.homing.triggerDirection == DIRECTION_POSITIVE)
				{
					/*	finished */
					pPathGenerator->moveCommand = MOVE_COMMAND_STOP;
					pPathGenerator->deceleration = p->param.deceleration;
					pIntern->step = 250;
				}
				else
				{
					/*	turn direction */
					pPathGenerator->moveCommand = MOVE_COMMAND_VELOCITY;
					pPathGenerator->setSpeed = -ABS(p->param.homing.speed2);
				}
			}

			if (pPathGenerator->outputSpeed < 0)
			{
				if (p->param.homing.triggerDirection == DIRECTION_NEGATIVE)
				{
					/*	finished */
					pPathGenerator->moveCommand = MOVE_COMMAND_STOP;
					pPathGenerator->deceleration = p->param.deceleration;
					pIntern->step = 250;
				}
				else
				{
					/*	turn direction */
					pPathGenerator->moveCommand = MOVE_COMMAND_VELOCITY;
					pPathGenerator->setSpeed = ABS(p->param.homing.speed2);
				}
			}
		}
		break;

	case 250:
		/*	wait till still */
		if (pPathGenerator->motionState == MOTION_STATE_STANDSTILL) pIntern->step = 260;
		break;

/***********************************************************************************************
	DIRECT_HOMING
************************************************************************************************/
	case 260:

		/*	set intern position inside path generator to actual position */
		PathGeneratorSetPosition(pPathGenerator, p->param.position);

		#ifdef ENCODER_POSITION
			ConvertPositionInitialize(pEncoder2units,p->init.encoderIncrements,p->init.units,p->init.reverseDirection,
				ENCODER_POSITION,p->param.position);
		#endif

		RESET_OUTPUT

		/*	set flag */
		p->info.homingOk = 1;
		/*	clear flag */
		p->cmd.homing = 0;
		pIntern->step=100;
		break;

	case 1000:
		/*	clear all commands, except of cmd.power */
		p->cmd.homing = 0;
		p->cmd.absolute = 0;
		p->cmd.additive = 0;
		p->cmd.cyclicPosition = 0;
		p->cmd.velocity = 0;
		p->cmd.acknowledge = 0;
		p->cmd.stop = 0;

		/*	stop movement */
		pPathGenerator->moveCommand = MOVE_COMMAND_STOP;
		pPathGenerator->deceleration = p->param.deceleration;

		/*	display error message */
		if(p->info.status == ERR_CONTROLLER_OFF)
		{
			strncpy(p->info.errorText,"It is not possible to make any movement because the controller is OFF ",sizeof(p->info.errorText));
		}

		if(p->info.status == ERR_WRONG_UNITS)
		{
			strncpy(p->info.errorText,"Value of \"init.units\" must be >= 1000",sizeof(p->info.errorText));
		}

		if(p->info.status == ERR_NEGATIVE_LIMIT_SWITCH_CLOSED)
		{
			strncpy(p->info.errorText,"Negative limit switch was activated",sizeof(p->info.errorText));
		}

		if(p->info.status == ERR_NEGATIVE_SW_LIMIT_REACHED)
		{
			strncpy(p->info.errorText,"Negative SW limit was reached",sizeof(p->info.errorText));
		}

		if(p->info.status == ERR_DRIVE_NOT_READY)
		{
			strncpy(p->info.errorText,"Drive is not ready",sizeof(p->info.errorText));
		}

		if(p->info.status == ERR_OVER_CURRENT)
		{
			strncpy(p->info.errorText,"Motor overcurrent",sizeof(p->info.errorText));
		}

		if(p->info.status == ERR_OVER_TEMPERATURE)
		{
			strncpy(p->info.errorText,"Motor overtemperature",sizeof(p->info.errorText));
		}

		if(p->info.status == ERR_POSITIVE_LIMIT_SWITCH_CLOSED)
		{
			strncpy(p->info.errorText,"Positive limit switch was activated",sizeof(p->info.errorText));
		}

		if(p->info.status == ERR_POSITIVE_SW_LIMIT_REACHED)
		{
			strncpy(p->info.errorText,"Positive SW limit was reached",sizeof(p->info.errorText));
		}

		if(p->info.status == ERR_STALL)
		{
			strncpy(p->info.errorText,"Stall detected",sizeof(p->info.errorText));
		}

		if(p->info.status == ERR_POWER_SUPPLY_ERROR)
		{
			strncpy(p->info.errorText,"Power supply problem",sizeof(p->info.errorText));
		}

		if(p->info.status == ERR_UNDER_VOLTAGE)
		{
			strncpy(p->info.errorText,"Low supply voltage",sizeof(p->info.errorText));
		}

		if(p->info.status == ERR_OVER_VOLTAGE)
		{
			strncpy(p->info.errorText,"High supply voltage",sizeof(p->info.errorText));
		}

		if(p->info.status == ERR_LAG_ERROR)
		{
			strncpy(p->info.errorText,"Lag error exceeded \"init.maxLagError\"",sizeof(p->info.errorText));
		}

		if(p->info.status == ERR_ENCODER_SUPPLY)
		{
			strncpy(p->info.errorText,"Encoder supply error",sizeof(p->info.errorText));
		}

		if(p->info.status == ERR_WRONG_TASK_TIME)
		{
			strncpy(p->info.errorText,"Value of \"init.taskTime\" must be between 0 and 1 sec" ,sizeof(p->info.errorText));
		}

		if(p->info.status == ERR_LOW_DC_BUS_VOLTAGE)
		{
			strncpy(p->info.errorText,"Low DC BUS voltage",sizeof(p->info.errorText));
		}

		if(p->info.status == ERR_WRONG_ENCODER_INCREMENTS)
		{
			strncpy(p->info.errorText,"Value of \"init.encoderIncrements\" must be > 0",sizeof(p->info.errorText));
		}

		if(p->info.status == ERR_DRV_NOT_OK)
		{
			strncpy(p->info.errorText,"\"DrvOk\" must be \"TRUE\"",sizeof(p->info.errorText));
		}
		pIntern->step++;
		break;

	case 1001:
		/*	wait till movement stopped */
		if (p->info.moveActive == 0)
		{
			pIntern->step++;
		}
		break;

		pIntern->step++;
		break;

	case 1002:
		/*	if controller should be switched off */
		if	(p->cmd.power == 0 || p->info.status == ERR_OVER_TEMPERATURE || p->info.status == ERR_OVER_CURRENT ||
			p->info.status == ERR_LAG_ERROR || p->info.status == ERR_STALL)
		{
			/*	switch controller off */
			p->info.powerOn = 0;
		}

		/*	wait for acknowledgement */
		if (p->cmd.acknowledge)
		{
			pIntern->step++;
		}
		break;

	case 1003:

		/*	acknowledge error form path generator */
		PathGeneratorResetError(pPathGenerator);

		/*	clear commands */
		p->cmd.acknowledge = 0;
		//p->info.status = 0;
		strcpy(p->info.errorText,"");

		pIntern->step = 1010;
		break;
```

#### every_cycle.h
```c
/***********************************************************************************************
	THINGS TO DO EVERY CYCLE
************************************************************************************************/
	if (!p->info.initialized) return;

/***********************************************************************************************
	PATH GENERATOR
************************************************************************************************/
	PathGenerator(pPathGenerator);

/***********************************************************************************************
	ACTUAL POSITION, LAG ERROR
************************************************************************************************/
#ifdef ENCODER_USED
	p->info.position = ConvertPosition(pEncoder2units, ENCODER_POSITION);
	p->info.lagError = pPathGenerator->outputPosition - p->info.position;
#else
	p->info.position = pPathGenerator->outputPosition;
#endif

/***********************************************************************************************
	ACTUAL SPEED
************************************************************************************************/
#ifdef ENCODER_USED
	pActualSpeed->actPosition = p->info.position;
	ActualSpeed(pActualSpeed);
	p->info.speed = pActualSpeed->actSpeed;
#else
	p->info.speed = pPathGenerator->outputSpeed;
#endif

/***********************************************************************************************
	FOR HOMING
************************************************************************************************/
	pIntern->oldReferenceSwitch = p->IOMapping.referenceSwitch;

/***********************************************************************************************
	DETERMINE MoveActive
************************************************************************************************/
	pMoveActive->motionState = pPathGenerator->motionState;
	MoveActive(pMoveActive);
	p->info.moveActive = pMoveActive->moveActive;

/***********************************************************************************************
	Set DriveEnable
************************************************************************************************/
	pIOMapping->DriveEnable = p->info.powerOn;
```

#### auxiliaries.h
```c
#ifndef _MOTORKY_AUXILIARIES_
#define _MOTORKY_AUXILIARIES_

#include <bur/plctypes.h>

#define INT_MAXVALUE	0x7FFF
#define DINT_MAXVALUE	0x7FFFFFFF
#define DEFAULT_SPEED			1000
#define DEFAULT_ACCELERATION	5000
/*
#define BIT_SET(value,bit)		value|=1<<(bit)
#define BIT_GET(value,bit)  	(value&(1<<(bit)))?1:0
#define BIT_CLR(value,bit)		value&=~(1<<(bit))
*/

void ActualSpeedInitialize(Motorky_ActualSpeed *pActualSpeed, REAL taskTime, REAL filterTime);
void ActualSpeed(Motorky_ActualSpeed *pActualSpeed);

void ConvertPositionInitialize(Motorky_ConvertPosition *pConvertPosition, DINT inputScale, DINT outputScale, BOOL reverseDirection,
	INT input, DINT output);
DINT ConvertPosition(Motorky_ConvertPosition *pConvertPosition, INT input);
DINT ConvertTime(REAL realVar);
void MoveActiveInitialize(Motorky_MoveActive *pMoveActive, REAL TaskTime, REAL SettleTime);
void MoveActive(Motorky_MoveActive *pMoveActive);
void TOFInitialize(Motorky_TOF *pTOF, REAL TaskTime, REAL PT);
void TOF(Motorky_TOF *pTOF);
void PIDInitialize(Motorky_PID *pPID, REAL Kp, REAL Tn, REAL TaskTime, DINT Y_max, DINT Y_min);
void PID(Motorky_PID *pPID);

#endif /* _MOTORKY_AUXILIARIES_ */
```

#### auxiliaries.c
```c
#include <motorky.h>
#include "auxiliaries.h"

void ActualSpeedInitialize(Motorky_ActualSpeed *pActualSpeed, REAL taskTime, REAL filterTime)
{
	pActualSpeed->taskTime = ConvertTime(taskTime);
	pActualSpeed->filterTime = ConvertTime(filterTime);

	/*	calculate FIFO size */
	if (pActualSpeed->taskTime > 0)
	{
		pActualSpeed->FIFOsize = pActualSpeed->filterTime/pActualSpeed->taskTime;
	}

	/* correct FIFOsize */
	if (pActualSpeed->FIFOsize <= 0) pActualSpeed->FIFOsize = 1;
	if (pActualSpeed->FIFOsize > SPEED_FIFO_UBOUND+1) pActualSpeed->FIFOsize = SPEED_FIFO_UBOUND+1;

	/* calculate FIFO length in us */
	pActualSpeed->filterTime = pActualSpeed->taskTime*pActualSpeed->FIFOsize;

	/* initialize FIFO with actual position */
/*	INT index1;
	for (index1=0; index1<=SPEED_FIFO_UBOUND; index1++)
	{
		pActualSpeed->positionFIFO[index1] = pActualSpeed->actPosition;
	}*/
}

void ActualSpeed(Motorky_ActualSpeed *pActualSpeed)
{
	DINT *pPosition;

	/*	increase FIFO index */
	if (++pActualSpeed->FIFOindex >= pActualSpeed->FIFOsize)
	{
		pActualSpeed->FIFOindex = 0;
	}

	/* get pointer to old value */
	pPosition = pActualSpeed->positionFIFO + pActualSpeed->FIFOindex;

	/*	calculate position difference */
	pActualSpeed->positionDifference = pActualSpeed->actPosition - *pPosition;

	/*	store new value to FIFO */
	*pPosition = pActualSpeed->actPosition;

	/* compute speed */
	pActualSpeed->actSpeed = (long long)pActualSpeed->positionDifference*1000000/pActualSpeed->filterTime;

}

void ConvertPositionInitialize(Motorky_ConvertPosition *pConvertPosition, DINT inputScale, DINT outputScale,
	BOOL reverseDirection, INT input, DINT output)
{
	pConvertPosition->inputScale = inputScale;
	pConvertPosition->outputScale = outputScale;
	pConvertPosition->reverseDirection = reverseDirection;

	pConvertPosition->input = input;
	pConvertPosition->output = output;
	pConvertPosition->integral = 0;
}

/*	this FUB converts units to steps */
DINT ConvertPosition(Motorky_ConvertPosition *pConvertPosition, INT input)
{
	long long integral;

	if (pConvertPosition->inputScale == 0) return 0;

	/*	difference */
	pConvertPosition->dInput = input - pConvertPosition->input;

	/*	store old value */
	pConvertPosition->input = input;

	/*	if there was an change, do computation */
	if (pConvertPosition->dInput != 0)
	{
		/*	reverse direction? */
		if (pConvertPosition->reverseDirection)
		{
			pConvertPosition->dInput = -pConvertPosition->dInput;
		}

		/*	copy value */
		integral = pConvertPosition->integral;

		/*	integrate */
		integral += (long long)pConvertPosition->dInput*pConvertPosition->outputScale;

		/*	modify output */
		pConvertPosition->output += integral/pConvertPosition->inputScale;

		/*	and compute rest */
		integral %= pConvertPosition->inputScale;

		/*	store back */
		pConvertPosition->integral = integral;
	}

	return pConvertPosition->output;
}

DINT ConvertTime(REAL realVar)
{
	if (realVar >=0 && realVar <= DINT_MAXVALUE/1000000)
	{
		return (1000000*realVar+0.5);
	}
	else
	{
		/* error */
		return -1;
	}
}

void MoveActiveInitialize(Motorky_MoveActive *pMoveActive, REAL TaskTime, REAL SettleTime)
{
	pMoveActive->taskTime = ConvertTime(TaskTime);
	pMoveActive->settleTime = ConvertTime(SettleTime);
}

void MoveActive(Motorky_MoveActive *pMoveActive)
{
	if (pMoveActive->motionState == MOTION_STATE_STANDSTILL)
	{
		/*	increase timer */
		pMoveActive->settleTimer += pMoveActive->taskTime;

		if (pMoveActive->settleTimer > pMoveActive->settleTime)
		{
			/*	limit timer */
			pMoveActive->settleTimer = pMoveActive->settleTime;
			/*	position reached */
			pMoveActive->moveActive = 0;
		}
	}
	else
	{
		/*	reset timer */
		pMoveActive->settleTimer = 0;
		/*	position not reached */
		pMoveActive->moveActive = 1;
	}
}

void TOFInitialize(Motorky_TOF *pTOF, REAL TaskTime, REAL PT)
{
	pTOF->PT = ConvertTime(PT)/ConvertTime(TaskTime);
}

void TOF(Motorky_TOF *pTOF)
{
	if (pTOF->IN == 1)
	{
		pTOF->Q = 1;
		pTOF->ET = 0;
	}
	else
	{
		if (++pTOF->ET > pTOF->PT) pTOF->ET = pTOF->PT;
	}

	if (pTOF->ET == pTOF->PT)
	{
		pTOF->Q = 0;
	}
	else
	{
		pTOF->Q = 1;
	}
}

void PIDInitialize(Motorky_PID *pPID, REAL Kp, REAL Tn, REAL TaskTime, DINT Y_max, DINT Y_min)
{
	pPID->Yi = 0;
	pPID->Yi_sum = 0;
	pPID->Y = 0;

	/*	scale REALs to DINT */
	pPID->Kp = INT_MAXVALUE * Kp;

	/*	compute divisor of Kp */
	pPID->Ki = Tn/TaskTime;

	pPID->Y_max = Y_max;
	pPID->Y_min = Y_min;
}

void PID(Motorky_PID *pPID)
{
	if (pPID->enable)
	{
		/* 	compute deviation */
		pPID->e = pPID->W - pPID->X;

		/*	compute proportional action */
		pPID->Yp = ((long long)pPID->Kp*pPID->e)/INT_MAXVALUE;

		/*	compute integral action */
		if (pPID->Ki > 0)
		{
			pPID->Yi_sum += pPID->Yp;
			pPID->Yi += pPID->Yi_sum/pPID->Ki;
			pPID->Yi_sum %= pPID->Ki;
		}
		else
		{
			/*	integral action is not used */
			pPID->Yi = 0;
			pPID->Yi_sum = 0;
		}
	}
	else
	{
		/*	no output */
		pPID->Yp = 0;
		pPID->Yi = 0;
		pPID->Yi_sum = 0;
	}

	/*	compute output value */
	pPID->Ytotal = pPID->Yp + pPID->Yi;

	/*	limit output */
	if (pPID->Ytotal > pPID->Y_max)
	{
		pPID->Ylim = pPID->Y_max;
	}
	else if (pPID->Ytotal < pPID->Y_min)
	{
		pPID->Ylim = pPID->Y_min;
	}
	else
	{
		pPID->Ylim = pPID->Ytotal;
	}

	/*	ramp limiter - at this time not implemented */
	pPID->Y = pPID->Ylim;

	/*	anti-windup */
	pPID->Ywindup = pPID->Y - pPID->Ytotal;
	pPID->Yi += pPID->Ywindup;
}
```

### Library Logical/Libraries/Atrima (IEC)

#### Types.typ - Exported data types
```iecst
TYPE
	StateDoor :
		(
		stateDoorLocked,
		stateDoorStopRequest,
		stateDoorUnlocked
		);
	ModeZone :
		(
		modeZoneOff,
		modeZoneManual,
		modeZoneAuto
		);
	MoveType :
		(
		moveTypeNo,
		moveTypeGoHome,
		moveTypeGoToTable,
		moveTypeGoForSeparator,
		moveTypePutSeparatorOnPallet,
		moveTypeVerticalOffset,
		moveTypePlaceFirstHalf,
		moveTypePlaceSecondHalf,
		moveTypeRelativeHorizontalOffset,
		moveTypeVerticalOffset2,
		moveTypeEndGoToTable
		);
END_TYPE
```

#### Atrima.fun - Exported functions and function blocks
```iecst
FUNCTION_BLOCK Comau
	VAR_INPUT
		DriveOn : BOOL;
		NoDriveOff : BOOL;
		Start : BOOL;
		NoHold : BOOL;
		CancelAlarm : BOOL;
		SafetySpeed : BOOL;
		MakeMove : BOOL;
		MoveType : MoveType;
		ProductType : USINT;
		NbOfLayers : USINT;
		diSensorBellowHead : BOOL;
		RawInput1 : UDINT;
		RawInput2 : UDINT;
	END_VAR
	VAR_OUTPUT
		NoAlarm : BOOL;
		DriveOnStatus : BOOL;
		Start_NoHoldPrgMove : BOOL;
		Remote : BOOL;
		SafetySpeedActive : BOOL;
		ProgrammingMode : BOOL;
		HeartBit : BOOL;
		MoveDone : BOOL;
		IsItSafeToGoHome : BOOL;
		Error : BOOL;
		ErrorHoldPressed : BOOL;
		RawOutput1 : UDINT;
		RawOutput2 : UDINT;
	END_VAR
	VAR
		moveActive : BOOL;
		checkMoveType : MoveType;
		checkProductType : USINT;
		checkNbOfLayers : USINT;
		startMove : BOOL;
		tmpRawOutput : UDINT;
		state : INT;
		MTBasicsPWM_0 : MTBasicsPWM;
	END_VAR
END_FUNCTION_BLOCK

FUNCTION_BLOCK DoorLogic
	VAR_INPUT
		diOpenButton : BOOL;
		diCloseButton : BOOL;
		modeZone : ModeZone;
		diDoorLocked : BOOL;
	END_VAR
	VAR_OUTPUT
		doUnlockDoors : BOOL;
		doLED : BOOL;
		stopRequest : BOOL;
	END_VAR
	VAR
		stateDoor : StateDoor;
		MTBasicsPWM_0 : MTBasicsPWM;
	END_VAR
END_FUNCTION_BLOCK
```

#### Atrima.st
```iecst
FUNCTION_BLOCK Comau

	//RawInput1
	NoAlarm				:= RawInput1.0;
	DriveOnStatus		:= RawInput1.1;
	Start_NoHoldPrgMove	:= RawInput1.2;
	Remote 				:= RawInput1.3;
	SafetySpeedActive	:= RawInput1.10;
	ProgrammingMode		:= RawInput1.11;
	HeartBit			:= RawInput1.15;

	//RawInput2
	moveActive := RawInput2.0;
	IsItSafeToGoHome := RawInput2.1;
	//MoveCheckOk := RawInput2.2;
	checkMoveType := UDINT_TO_USINT(SHR(RawInput2, 8));
	checkProductType := UDINT_TO_USINT(SHR(RawInput2, 16));
	checkNbOfLayers	:= UDINT_TO_USINT(SHR(RawInput2, 24));

	IF NOT MakeMove THEN
		state := 0;
		MoveDone := FALSE;
		startMove := FALSE;
		Error := FALSE;
		ErrorHoldPressed := FALSE;
	END_IF

	CASE state OF
		0:
			IF MakeMove THEN
				state := state + 1;
			END_IF

		1:
			IF moveActive THEN
				IF MoveType = checkMoveType AND ProductType = checkProductType AND NbOfLayers = checkNbOfLayers THEN
					state := state + 1;
				ELSE
					Error := TRUE;
					state := 5;
				END_IF
			ELSE
				state := state + 1;
			END_IF

		2:
			MTBasicsPWM_0(Enable :=  TRUE, Period := 1, DutyCycle := 50);
			Start := MTBasicsPWM_0.Out;

			IF Start_NoHoldPrgMove THEN
				Start := FALSE;
				state := state + 1;
			END_IF

		3:
			startMove := TRUE;

			IF moveActive THEN
				startMove := FALSE;
				state := state + 1;
			END_IF

		4:
			IF NOT moveActive THEN
				MoveDone := TRUE;
				state := state + 1;
			END_IF

			IF NOT Start_NoHoldPrgMove THEN
				ErrorHoldPressed := TRUE;
				state := 5;
			END_IF
		5:

	END_CASE;

	//RawOutput1
	tmpRawOutput := 0;
	tmpRawOutput.0 := DriveOn;
	tmpRawOutput.1 := NoDriveOff;
	tmpRawOutput.2 := Start;
	tmpRawOutput.3 := NoHold;
	tmpRawOutput.8 := CancelAlarm;
	tmpRawOutput.9 := SafetySpeed;
	RawOutput1 := tmpRawOutput;

	//RawOutput2
	tmpRawOutput := 0;
	tmpRawOutput.0 := startMove;
	tmpRawOutput.1 := diSensorBellowHead;
	tmpRawOutput := tmpRawOutput OR SHL(DINT_TO_UDINT(MoveType),8);
	tmpRawOutput := tmpRawOutput OR SHL(USINT_TO_UDINT(ProductType),16);
	tmpRawOutput := tmpRawOutput OR SHL(USINT_TO_UDINT(NbOfLayers),24);
	RawOutput2 := tmpRawOutput;

END_FUNCTION_BLOCK

FUNCTION_BLOCK DoorLogic

	diDoorLocked;

	CASE stateDoor OF

		stateDoorLocked:

			stopRequest := FALSE;

			IF diOpenButton THEN
				stateDoor := stateDoorStopRequest;
			END_IF

			doLED := FALSE;
			doUnlockDoors := FALSE;

		stateDoorStopRequest:

			stopRequest := TRUE;

			IF modeZone <> modeZoneAuto THEN
				stateDoor := stateDoorUnlocked;
			END_IF

			doLED := TRUE;
			doUnlockDoors := FALSE;

		stateDoorUnlocked:

			IF diCloseButton THEN
				stateDoor := stateDoorLocked;
			END_IF

			MTBasicsPWM_0(Enable := 1, DutyCycle := 50, Period := 1);

			doLED := MTBasicsPWM_0.Out;
			doUnlockDoors := TRUE;

	END_CASE

END_FUNCTION_BLOCK
```

### Library Logical/Libraries/Misc (IEC)

#### Types.typ - Exported data types
```iecst
TYPE
	StateDoor :
		(
		stateDoorLocked,
		stateDoorStopRequest,
		stateDoorUnlocked
		);
	ModeZone :
		(
		modeZoneNotReadyToStart,
		modeZoneManual,
		modeZoneAuto
		);
END_TYPE
```

#### Misc.fun - Exported functions and function blocks
```iecst
FUNCTION_BLOCK DoorLogic
	VAR_INPUT
		buttonToOpen : BOOL;
		buttonToClose : BOOL;
		modeZone : ModeZone;
		doorLocked : BOOL;
	END_VAR
	VAR_OUTPUT
		unlockDoors : BOOL;
		LED : BOOL;
		stopRequest : BOOL;
	END_VAR
	VAR
		stateDoor : StateDoor;
		MTBasicsPWM_0 : MTBasicsPWM;
	END_VAR
END_FUNCTION_BLOCK
```

#### Misc.st
```iecst
FUNCTION_BLOCK DoorLogic

	CASE stateDoor OF

		stateDoorLocked:

			stopRequest := FALSE;

			IF buttonToOpen THEN
				stateDoor := stateDoorStopRequest;
			END_IF

			LED := FALSE;
			unlockDoors := FALSE;

		stateDoorStopRequest:

			stopRequest := TRUE;

			IF modeZone <> modeZoneAuto THEN
				stateDoor := stateDoorUnlocked;
			END_IF

			LED := TRUE;
			unlockDoors := FALSE;

		stateDoorUnlocked:

			IF buttonToClose THEN
				stateDoor := stateDoorLocked;
			END_IF

			MTBasicsPWM_0(Enable := 1, DutyCycle := 50, Period := 1);

			LED := MTBasicsPWM_0.Out;
			unlockDoors := TRUE;

	END_CASE

END_FUNCTION_BLOCK
```

### pallet_magazine.typ
```iecst
TYPE
	PalletStatus :
		(
		palletNotPresent,
		palletPresent,
		palletMoving
		);
	ModeMagazine :
		(
		modeMagazineNotReadyToStart,
		modeMagazineManual,
		modeMagazineAuto
		);
END_TYPE
```

### pallet_magazine.var
```iecst
VAR
	acknowledgeImageMagazine : ARRAY[0..39] OF BOOL;
	alarmImageMagazine : ARRAY[0..39] OF BOOL;
	cmdMagazineAuto : BOOL; (*VISU:switches pallet magazine to automatic mode*)
	cmdMagazineManual : BOOL;
	magazineEmpty : BOOL;
	modeZoneMagazine : ModeZone;
END_VAR
```

### Program Logical/plc/pallet_magazine/pallet_magazine (IEC) - pallet magazine control

#### Main.st
```iecst
(*Control OF pallet magazine, also called "zásobník palet" nebo "stohovač" *)

PROGRAM _INIT

END_PROGRAM

PROGRAM _CYCLIC

	modeZoneMagazineOld := modeZoneMagazine;

	readyToStart := NOT diMagazineEDM;

	IF cpuIsSimulated THEN
		readyToStart := TRUE;
	END_IF

	IF NOT readyToStart THEN
		modeZoneMagazine := modeZoneOff;
	END_IF

	CASE modeZoneMagazine OF

		modeZoneOff: //the automat is not ready to start

			IF readyToStart THEN
				modeZoneMagazine := modeZoneManual;
			END_IF
			cmdMagazineManual := FALSE;
			cmdMagazineAuto := FALSE;
			magazineEmpty := FALSE;

		modeZoneManual:

			IF modeZoneMagazineOld <> modeZoneManual THEN
			END_IF

			IF (NOT alarmInZoneMagazine OR cpuIsSimulated) AND (cmdMagazineAuto OR TP_Start.Q) THEN
				modeZoneMagazine := modeZoneAuto;
				stateAuto := stateAutoUndefined;
			END_IF
			cmdMagazineManual := FALSE;

			magazineEmpty := FALSE;

		modeZoneAuto:

			IF (alarmInZoneMagazine AND NOT cpuIsSimulated) OR cmdMagazineManual THEN
				modeZoneMagazine := modeZoneManual;
			END_IF
			cmdMagazineAuto := FALSE;

			CASE stateAuto OF

				stateAutoUndefined:

					cmdUp := FALSE;
					IF stateMagazine = stateUpperPosition THEN
						stateAuto := stateAutoWaitForNoPallet;
					ELSIF stateMagazine = stateMiddlePosition THEN
						stateAuto := stateAutoCloseArms;
					ELSIF stateMagazine = stateLowerPosition THEN
						stateAuto := stateAutoOpenArms;
					ELSE
						cmdUp := TRUE;
					END_IF

				stateAutoWaitForNoPallet:

					IF statePalletP12 = palletNotPresent AND NOT magazineEmpty THEN
						stateAuto := stateAutoMoveToLowerPosition;
					END_IF

				stateAutoMoveToLowerPosition:

					cmdDown := TRUE;
					stateAuto := stateAutoWaitForLowerPosition;

				stateAutoWaitForLowerPosition:

					IF stateMagazine = stateLowerPosition THEN
						stateAuto := stateAutoOpenArms;
					END_IF

				stateAutoOpenArms:

					closeArms := FALSE;
					stateAuto := stateAutoWaitForOpenedArms;

				stateAutoWaitForOpenedArms:

					IF stateArms = stateArmsOpened THEN
						stateAuto := stateAutoMoveToMiddlePosition;
					END_IF

				stateAutoMoveToMiddlePosition:

					cmdUp := TRUE;
					stateAuto := stateAutoWaitForMiddlePosition;

				stateAutoWaitForMiddlePosition:

					IF stateMagazine = stateMiddlePosition THEN
						stateAuto := stateAutoCloseArms;
					END_IF

				stateAutoCloseArms:

					closeArms := TRUE;
					stateAuto := stateAutoWaitForClosedArms;

				stateAutoWaitForClosedArms:

					IF stateArms = stateArmsClosed THEN
						cmdUp := TRUE;
						stateAuto := stateAutoMoveToUpperPosition;
					END_IF

				stateAutoMoveToUpperPosition:

					IF stateMagazine = stateUpperPosition THEN
						stateAuto := stateAutoDetectPalletOnConveyor;
					END_IF

				stateAutoDetectPalletOnConveyor:

					IF statePalletP12 = palletNotPresent THEN
						magazineEmpty := TRUE;
					END_IF
					stateAuto := stateAutoWaitForNoPallet;

			END_CASE

	END_CASE;

	//horizontal arms movement
	HorizontalArmsControl;

	//vertical arms movement
	VerticalArmsControl;

	//conveyor P12
	//ConveyorP12Control;

	TON_PalletOnConveyorP12(IN := diPalletOnConveyorP12, PT := T#50ms);

	//detect pallet on conveyor
	IF TON_PalletOnConveyorP12.Q AND stateMagazine = stateUpperPosition AND statePalletP12 = palletNotPresent THEN
		statePalletP12 := palletPresent;
	END_IF

	//LED P11
	IF diMagazineEDM THEN
		MTBasicsPWM_0.DutyCycle := 50;
	ELSE
		MTBasicsPWM_0.DutyCycle := 0;
	END_IF

	MTBasicsPWM_0(Enable := 1, Period := 1);
	doLedP11 := MTBasicsPWM_0.Out;

	TP_Start(IN := diActivateMagazineSafetyCircuits AND modeZonePalletization = modeZoneAuto, PT := T#1s);

	alarmImageMagazine[1] := NOT lightCurtainP11;
	alarmImageMagazine[6] := NOT diMotorProtectionP11;

END_PROGRAM
```

#### Types.typ - Local data types
```iecst
TYPE
	StateAuto :
		(
		stateAutoUndefined,
		stateAutoWaitForNoPallet,
		stateAutoMoveToLowerPosition,
		stateAutoWaitForLowerPosition,
		stateAutoOpenArms,
		stateAutoWaitForOpenedArms,
		stateAutoMoveToMiddlePosition,
		stateAutoWaitForMiddlePosition,
		stateAutoCloseArms,
		stateAutoWaitForClosedArms,
		stateAutoMoveToUpperPosition,
		stateAutoDetectPalletOnConveyor
		);
	StateMagazine :
		(
		stateMagazineUndefined,
		stateMoveToUpperPosition,
		stateUpperPosition,
		stateMoveLowerToMiddlePosition,
		stateMiddlePosition,
		stateMoveToLowerPosition,
		stateLowerPosition
		);
	StateArms :
		(
		stateArmsInit,
		stateArmsOpening,
		stateArmsOpened,
		stateArmsClosing,
		stateArmsClosed
		);
END_TYPE
```
